KUKA KRL program: EPS_2_25362_MH4A_A_20251103083058.src

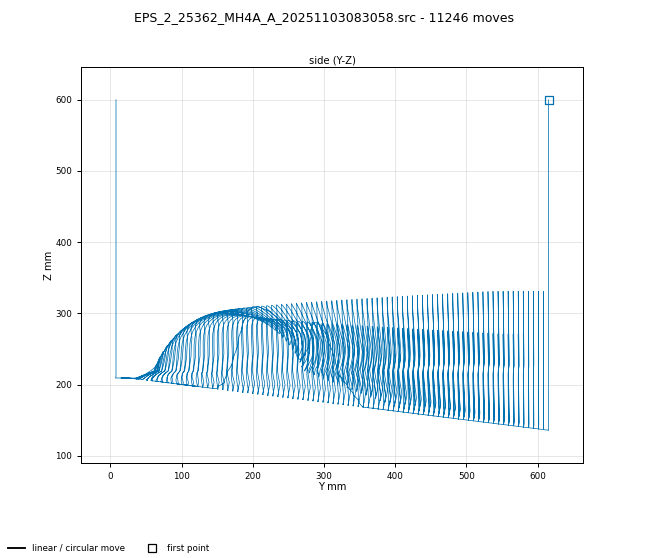
[picture p0: tool path of EPS_2_25362_MH4A_A_20251103083058.src, 11246 of 11248 moves have a stored position in this frame; points joined in program order, loops and branches not executed]
&ACCESS RVP
&REL 4
&COMMENT QRS 19112012
&PARAM EDITMASK = *
DEF PART()
EXT BAS (BAS_COMMAND :IN,REAL :IN )
INT I
BAS (#INITMOV,0 )

;KUKA QRS Post kuka4.cps  Date:22-06-2017 !

File_ID=2901

QRS_PRE_INIT()

;Init var - Until changes are made in qrs_pre_init
Outlet_Square_prg=0
Inlet_1_Square_prg=0
Inlet_2_Square_prg=0
Inlet_3_Square_prg=0
Inlet_4_Square_prg=0
Inlet_5_Square_prg=0

Outlet_1={X 0.000, Y 537.380, Z 230.500, B 0.000, E1 0.000 }
Inlet_1={X 0.000, Y 549.320, Z 220.500, B 0.000, E1 270.000 }
Outlet_1_type=201
Inlet_1_type=101
;QRS#1=Sidecore dimensions
;QRS#2=200-8" PVC SDR 35
;QRS#3=100-4" PVC SDR 28
;QRS#4=
;QRS#5=
;QRS#6=
;QRS#7=
;QRS#8=
;QRS#9=12-08 PSX
;QRS#10=8QRS PSX
;QRS#11=
;QRS#12=
;QRS#13=
;QRS#14=
;QRS#15=
;QRS#16=1220x127x610 2'
;QRS#17=EPS Height
;QRS#18=331
;QRS#19=*
;QRS#20= UPDATED VERSION 22-06-2017
;QRS#21=*
Outlet_Square=0100
Inlet_1_Square=045
Inlet_2_Square=0
Inlet_3_Square=0
Inlet_4_Square=0
Inlet_5_Square=0
Mill_Square=1
Outlet_Square_Prg=204
Inlet_1_Square_prg=201

QRS_INIT()

$ADVANCE=5

; T1
PTP {E1 173.59,E2 173.59}
PTP {X 0,Y 615.51,A -85,B 0,C 180,E1 173.59,E2 173.59,E3 0,E4 0,E5 0,E6 0}
QRS_SPEED_INIT()
LIN {X 0,Y 615.51,Z 600,A -85,B 0,C 180,E1 173.59,E2 173.59,E3 0,E4 0,E5 0,E6 0} C_VEL
LIN {X 0,Y 615.51,Z 145.871,A -85,B 0,C 180,E1 173.59,E2 173.59} C_VEL
LIN {X 0,Y 615.51,Z 137.691,A -85,B 0,C 180,E1 173.59,E2 173.59} C_VEL
LIN {X 0,Y 615.491,Z 135.691,A -85,B 0,C 180,E1 173.404,E2 173.404} C_VEL
LIN {X 0,Y 615.484,Z 135.694,A -85,B 0,C 180,E1 170.801,E2 170.801} C_VEL
LIN {X 0,Y 615.456,Z 135.696,A -85,B 0,C 180,E1 168.139,E2 168.139} C_VEL
LIN {X 0,Y 615.487,Z 135.702,A -85,B 0,C 180,E1 165.451,E2 165.451} C_VEL
LIN {X 0,Y 615.449,Z 135.697,A -85,B 0,C 180,E1 162.728,E2 162.728} C_VEL
LIN {X 0,Y 615.489,Z 135.692,A -85,B 0,C 180,E1 159.967,E2 159.967} C_VEL
LIN {X 0,Y 615.484,Z 135.699,A -85,B 0,C 180,E1 157.155,E2 157.155} C_VEL
LIN {X 0,Y 615.453,Z 135.696,A -85,B 0,C 180,E1 154.434,E2 154.434} C_VEL
LIN {X 0,Y 615.456,Z 135.699,A -85,B 0,C 180,E1 151.552,E2 151.552} C_VEL
LIN {X 0,Y 615.471,Z 135.698,A -85,B 0,C 180,E1 148.913,E2 148.913} C_VEL
LIN {X 0,Y 615.488,Z 135.688,A -85,B 0,C 180,E1 145.978,E2 145.978} C_VEL
LIN {X 0,Y 615.484,Z 135.703,A -85,B 0,C 180,E1 143.575,E2 143.575} C_VEL
LIN {X 0,Y 615.444,Z 135.698,A -85,B 0,C 180,E1 140.94,E2 140.94} C_VEL
LIN {X 0,Y 615.498,Z 135.7,A -85,B 0,C 180,E1 138.527,E2 138.527} C_VEL
LIN {X 0,Y 615.464,Z 135.694,A -85,B 0,C 180,E1 135.848,E2 135.848} C_VEL
LIN {X 0,Y 615.479,Z 135.693,A -85,B 0,C 180,E1 133.046,E2 133.046} C_VEL
LIN {X 0,Y 615.491,Z 135.7,A -85,B 0,C 180,E1 130.089,E2 130.089} C_VEL
LIN {X 0,Y 615.45,Z 135.7,A -85,B 0,C 180,E1 127.243,E2 127.243} C_VEL
LIN {X 0,Y 615.484,Z 135.692,A -85,B 0,C 180,E1 124.7,E2 124.7} C_VEL
LIN {X 0,Y 615.47,Z 135.694,A -85,B 0,C 180,E1 122.328,E2 122.328} C_VEL
LIN {X 0,Y 615.479,Z 135.696,A -85,B 0,C 180,E1 119.793,E2 119.793} C_VEL
LIN {X 0,Y 615.498,Z 135.691,A -85,B 0,C 180,E1 117.047,E2 117.047} C_VEL
LIN {X 0,Y 615.435,Z 135.7,A -85,B 0,C 180,E1 114.273,E2 114.273} C_VEL
LIN {X 0,Y 615.495,Z 135.693,A -85,B 0,C 180,E1 111.43,E2 111.43} C_VEL
LIN {X 0,Y 615.482,Z 135.696,A -85,B 0,C 180,E1 108.603,E2 108.603} C_VEL
LIN {X 0,Y 615.47,Z 135.692,A -85,B 0,C 180,E1 105.904,E2 105.904} C_VEL
LIN {X 0,Y 615.484,Z 135.7,A -85,B 0,C 180,E1 103.2,E2 103.2} C_VEL
LIN {X 0,Y 615.442,Z 135.7,A -85,B 0,C 180,E1 100.527,E2 100.527} C_VEL
LIN {X 0,Y 615.493,Z 135.691,A -85,B 0,C 180,E1 97.874,E2 97.874} C_VEL
LIN {X 0,Y 615.483,Z 135.695,A -85,B 0,C 180,E1 95.24,E2 95.24} C_VEL
LIN {X 0,Y 615.461,Z 135.695,A -85,B 0,C 180,E1 92.617,E2 92.617} C_VEL
LIN {X 0,Y 615.486,Z 135.699,A -85,B 0,C 180,E1 89.999,E2 89.999} C_VEL
LIN {X 0,Y 615.446,Z 135.697,A -85,B 0,C 180,E1 87.381,E2 87.381} C_VEL
LIN {X 0,Y 615.491,Z 135.699,A -85,B 0,C 180,E1 84.758,E2 84.758} C_VEL
LIN {X 0,Y 615.488,Z 135.689,A -85,B 0,C 180,E1 82.123,E2 82.123} C_VEL
LIN {X 0,Y 615.466,Z 135.698,A -85,B 0,C 180,E1 79.472,E2 79.472} C_VEL
LIN {X 0,Y 615.458,Z 135.7,A -85,B 0,C 180,E1 76.797,E2 76.797} C_VEL
LIN {X 0,Y 615.461,Z 135.695,A -85,B 0,C 180,E1 74.093,E2 74.093} C_VEL
LIN {X 0,Y 615.492,Z 135.7,A -85,B 0,C 180,E1 71.353,E2 71.353} C_VEL
LIN {X 0,Y 615.492,Z 135.689,A -85,B 0,C 180,E1 68.567,E2 68.567} C_VEL
LIN {X 0,Y 615.446,Z 135.698,A -85,B 0,C 180,E1 65.725,E2 65.725} C_VEL
LIN {X 0,Y 615.485,Z 135.697,A -85,B 0,C 180,E1 62.822,E2 62.822} C_VEL
LIN {X 0,Y 615.462,Z 135.696,A -85,B 0,C 180,E1 60.21,E2 60.21} C_VEL
LIN {X 0,Y 615.479,Z 135.693,A -85,B 0,C 180,E1 57.541,E2 57.541} C_VEL
LIN {X 0,Y 615.496,Z 135.688,A -85,B 0,C 180,E1 55.185,E2 55.185} C_VEL
LIN {X 0,Y 615.471,Z 135.7,A -85,B 0,C 180,E1 52.756,E2 52.756} C_VEL
LIN {X 0,Y 615.459,Z 135.7,A -85,B 0,C 180,E1 49.914,E2 49.914} C_VEL
LIN {X 0,Y 615.494,Z 135.693,A -85,B 0,C 180,E1 47.647,E2 47.647} C_VEL
LIN {X 0,Y 615.478,Z 135.695,A -85,B 0,C 180,E1 44.93,E2 44.93} C_VEL
LIN {X 0,Y 615.463,Z 135.695,A -85,B 0,C 180,E1 42.355,E2 42.355} C_VEL
LIN {X 0,Y 615.491,Z 135.695,A -85,B 0,C 180,E1 39.75,E2 39.75} C_VEL
LIN {X 0,Y 615.441,Z 135.699,A -85,B 0,C 180,E1 36.93,E2 36.93} C_VEL
LIN {X 0,Y 615.479,Z 135.698,A -85,B 0,C 180,E1 34.699,E2 34.699} C_VEL
LIN {X 0,Y 615.481,Z 135.692,A -85,B 0,C 180,E1 32.329,E2 32.329} C_VEL
LIN {X 0,Y 615.493,Z 135.842,A -85,B 0,C 180,E1 29.746,E2 29.746} C_VEL
LIN {X 0,Y 615.494,Z 144.518,A -85,B 0,C 180,E1 27.045,E2 27.045} C_VEL
LIN {X 0,Y 615.484,Z 153.55,A -85,B 0,C 180,E1 24.272,E2 24.272} C_VEL
LIN {X 0,Y 615.429,Z 162.982,A -85,B 0,C 180,E1 21.434,E2 21.434} C_VEL
LIN {X 0,Y 615.491,Z 172.39,A -85,B 0,C 180,E1 18.646,E2 18.646} C_VEL
LIN {X 0,Y 615.466,Z 181.817,A -85,B 0,C 180,E1 15.906,E2 15.906} C_VEL
LIN {X 0,Y 615.484,Z 191.214,A -85,B 0,C 180,E1 13.201,E2 13.201} C_VEL
LIN {X 0,Y 615.49,Z 200.624,A -85,B 0,C 180,E1 10.527,E2 10.527} C_VEL
LIN {X 0,Y 615.463,Z 210.021,A -85,B 0,C 180,E1 7.876,E2 7.876} C_VEL
LIN {X 0,Y 615.497,Z 214.015,A -85,B 0,C 180,E1 6.761,E2 6.761} C_VEL
LIN {X 0,Y 615.497,Z 223.447,A -85,B 0,C 180,E1 6.474,E2 6.474} C_VEL
LIN {X 0,Y 615.451,Z 232.476,A -85,B 0,C 180,E1 6.063,E2 6.063} C_VEL
LIN {X 0,Y 615.437,Z 240.486,A -85,B 0,C 180,E1 5.57,E2 5.57} C_VEL
LIN {X 0,Y 615.483,Z 248.518,A -85,B 0,C 180,E1 4.913,E2 4.913} C_VEL
LIN {X 0,Y 615.497,Z 254.668,A -85,B 0,C 180,E1 4.256,E2 4.256} C_VEL
LIN {X 0,Y 615.497,Z 259.516,A -85,B 0,C 180,E1 3.601,E2 3.601} C_VEL
LIN {X 0,Y 615.498,Z 263.25,A -85,B 0,C 180,E1 2.945,E2 2.945} C_VEL
LIN {X 0,Y 615.498,Z 267.23,A -85,B 0,C 180,E1 1.963,E2 1.963} C_VEL
LIN {X 0,Y 615.496,Z 268.964,A -85,B 0,C 180,E1 1.309,E2 1.309} C_VEL
LIN {X 0,Y 615.496,Z 270.004,A -85,B 0,C 180,E1 0.654,E2 0.654} C_VEL
LIN {X 0,Y 615.494,Z 270.384,A -85,B 0,C 180,E1 0,E2 0} C_VEL
LIN {X 0,Y 615.496,Z 270.105,A -85,B 0,C 180,E1 -0.654,E2 -0.654} C_VEL
LIN {X 0,Y 615.497,Z 269.165,A -85,B 0,C 180,E1 -1.309,E2 -1.309} C_VEL
LIN {X 0,Y 615.496,Z 267.536,A -85,B 0,C 180,E1 -1.963,E2 -1.963} C_VEL
LIN {X 0,Y 615.498,Z 263.663,A -85,B 0,C 180,E1 -2.945,E2 -2.945} C_VEL
LIN {X 0,Y 615.5,Z 259.011,A -85,B 0,C 180,E1 -3.765,E2 -3.765} C_VEL
LIN {X 0,Y 615.498,Z 254.03,A -85,B 0,C 180,E1 -4.42,E2 -4.42} C_VEL
LIN {X 0,Y 615.467,Z 247.759,A -85,B 0,C 180,E1 -5.077,E2 -5.077} C_VEL
LIN {X 0,Y 615.43,Z 240.602,A -85,B 0,C 180,E1 -5.653,E2 -5.653} C_VEL
LIN {X 0,Y 615.448,Z 232.615,A -85,B 0,C 180,E1 -6.146,E2 -6.146} C_VEL
LIN {X 0,Y 615.488,Z 223.109,A -85,B 0,C 180,E1 -6.576,E2 -6.576} C_VEL
LIN {X 0,Y 615.489,Z 213.97,A -85,B 0,C 180,E1 -6.856,E2 -6.856} C_VEL
LIN {X 0,Y 615.458,Z 204.468,A -85,B 0,C 180,E1 -9.531,E2 -9.531} C_VEL
LIN {X 0,Y 615.485,Z 195.061,A -85,B 0,C 180,E1 -12.195,E2 -12.195} C_VEL
LIN {X 0,Y 615.482,Z 185.648,A -85,B 0,C 180,E1 -14.887,E2 -14.887} C_VEL
LIN {X 0,Y 615.461,Z 176.24,A -85,B 0,C 180,E1 -17.614,E2 -17.614} C_VEL
LIN {X 0,Y 615.468,Z 167.99,A -85,B 0,C 180,E1 -20.034,E2 -20.034} C_VEL
LIN {X 0,Y 615.44,Z 158.569,A -85,B 0,C 180,E1 -22.847,E2 -22.847} C_VEL
LIN {X 0,Y 615.439,Z 151.492,A -85,B 0,C 180,E1 -24.994,E2 -24.994} C_VEL
LIN {X 0,Y 615.496,Z 143.116,A -85,B 0,C 180,E1 -27.545,E2 -27.545} C_VEL
LIN {X 0,Y 615.489,Z 135.697,A -85,B 0,C 180,E1 -29.794,E2 -29.794} C_VEL
LIN {X 0,Y 615.488,Z 135.698,A -85,B 0,C 180,E1 -32.458,E2 -32.458} C_VEL
LIN {X 0,Y 615.493,Z 135.7,A -85,B 0,C 180,E1 -34.815,E2 -34.815} C_VEL
LIN {X 0,Y 615.491,Z 135.699,A -85,B 0,C 180,E1 -37.242,E2 -37.242} C_VEL
LIN {X 0,Y 615.489,Z 135.698,A -85,B 0,C 180,E1 -40.088,E2 -40.088} C_VEL
LIN {X 0,Y 615.487,Z 135.7,A -85,B 0,C 180,E1 -42.353,E2 -42.353} C_VEL
LIN {X 0,Y 615.485,Z 135.698,A -85,B 0,C 180,E1 -45.069,E2 -45.069} C_VEL
LIN {X 0,Y 615.494,Z 135.701,A -85,B 0,C 180,E1 -47.919,E2 -47.919} C_VEL
LIN {X 0,Y 615.487,Z 135.701,A -85,B 0,C 180,E1 -50.249,E2 -50.249} C_VEL
LIN {X 0,Y 615.483,Z 135.698,A -85,B 0,C 180,E1 -53.064,E2 -53.064} C_VEL
LIN {X 0,Y 615.496,Z 135.696,A -85,B 0,C 180,E1 -55.299,E2 -55.299} C_VEL
LIN {X 0,Y 615.494,Z 135.699,A -85,B 0,C 180,E1 -57.669,E2 -57.669} C_VEL
LIN {X 0,Y 615.479,Z 135.7,A -85,B 0,C 180,E1 -60.207,E2 -60.207} C_VEL
LIN {X 0,Y 615.498,Z 135.696,A -85,B 0,C 180,E1 -62.953,E2 -62.953} C_VEL
LIN {X 0,Y 615.472,Z 135.812,A -85,B 0,C 180,E1 -63.76,E2 -63.76} C_VEL
LIN {X 0,Y 615.493,Z 150.876,A -85,B 0,C 180,E1 -66.443,E2 -66.443} C_VEL
LIN {X 0,Y 615.49,Z 167.065,A -85,B 0,C 180,E1 -69.269,E2 -69.269} C_VEL
LIN {X 0,Y 615.477,Z 183.238,A -85,B 0,C 180,E1 -72.042,E2 -72.042} C_VEL
LIN {X 0,Y 615.485,Z 199.394,A -85,B 0,C 180,E1 -74.773,E2 -74.773} C_VEL
LIN {X 0,Y 615.491,Z 215.538,A -85,B 0,C 180,E1 -77.469,E2 -77.469} C_VEL
LIN {X 0,Y 615.493,Z 220.864,A -85,B 0,C 180,E1 -78.326,E2 -78.326} C_VEL
LIN {X 0,Y 615.486,Z 234.201,A -85,B 0,C 180,E1 -78.556,E2 -78.556} C_VEL
LIN {X 0,Y 615.476,Z 247.357,A -85,B 0,C 180,E1 -78.923,E2 -78.923} C_VEL
LIN {X 0,Y 615.486,Z 259.131,A -85,B 0,C 180,E1 -79.383,E2 -79.383} C_VEL
LIN {X 0,Y 615.483,Z 270.56,A -85,B 0,C 180,E1 -79.971,E2 -79.971} C_VEL
LIN {X 0,Y 615.499,Z 282.008,A -85,B 0,C 180,E1 -80.718,E2 -80.718} C_VEL
LIN {X 0,Y 615.498,Z 291.247,A -85,B 0,C 180,E1 -81.463,E2 -81.463} C_VEL
LIN {X 0,Y 615.5,Z 299.645,A -85,B 0,C 180,E1 -82.289,E2 -82.289} C_VEL
LIN {X 0,Y 615.497,Z 307.688,A -85,B 0,C 180,E1 -83.258,E2 -83.258} C_VEL
LIN {X 0,Y 615.499,Z 313.417,A -85,B 0,C 180,E1 -84.101,E2 -84.101} C_VEL
LIN {X 0,Y 615.496,Z 318.868,A -85,B 0,C 180,E1 -85.086,E2 -85.086} C_VEL
LIN {X 0,Y 615.497,Z 323.137,A -85,B 0,C 180,E1 -86.071,E2 -86.071} C_VEL
LIN {X 0,Y 615.494,Z 325.396,A -85,B 0,C 180,E1 -86.726,E2 -86.726} C_VEL
LIN {X 0,Y 615.497,Z 327.23,A -85,B 0,C 180,E1 -87.381,E2 -87.381} C_VEL
LIN {X 0,Y 615.5,Z 328.606,A -85,B 0,C 180,E1 -88.036,E2 -88.036} C_VEL
LIN {X 0,Y 615.496,Z 330.173,A -85,B 0,C 180,E1 -89.345,E2 -89.345} C_VEL
LIN {X 0,Y 615.494,Z 330.389,A -85,B 0,C 180,E1 -89.999,E2 -89.999} C_VEL
LIN {X 0,Y 615.495,Z 329.581,A -85,B 0,C 180,E1 -91.308,E2 -91.308} C_VEL
LIN {X 0,Y 615.5,Z 328.609,A -85,B 0,C 180,E1 -91.962,E2 -91.962} C_VEL
LIN {X 0,Y 615.497,Z 327.236,A -85,B 0,C 180,E1 -92.617,E2 -92.617} C_VEL
LIN {X 0,Y 615.496,Z 324.353,A -85,B 0,C 180,E1 -93.6,E2 -93.6} C_VEL
LIN {X 0,Y 615.498,Z 320.446,A -85,B 0,C 180,E1 -94.583,E2 -94.583} C_VEL
LIN {X 0,Y 615.499,Z 315.411,A -85,B 0,C 180,E1 -95.569,E2 -95.569} C_VEL
LIN {X 0,Y 615.496,Z 308.87,A -85,B 0,C 180,E1 -96.583,E2 -96.583} C_VEL
LIN {X 0,Y 615.497,Z 301.143,A -85,B 0,C 180,E1 -97.544,E2 -97.544} C_VEL
LIN {X 0,Y 615.498,Z 293.057,A -85,B 0,C 180,E1 -98.37,E2 -98.37} C_VEL
LIN {X 0,Y 615.499,Z 283.183,A -85,B 0,C 180,E1 -99.197,E2 -99.197} C_VEL
LIN {X 0,Y 615.485,Z 272.002,A -85,B 0,C 180,E1 -99.944,E2 -99.944} C_VEL
LIN {X 0,Y 615.489,Z 261.047,A -85,B 0,C 180,E1 -100.526,E2 -100.526} C_VEL
LIN {X 0,Y 615.476,Z 248.567,A -85,B 0,C 180,E1 -101.038,E2 -101.038} C_VEL
LIN {X 0,Y 615.485,Z 236.118,A -85,B 0,C 180,E1 -101.4,E2 -101.4} C_VEL
LIN {X 0,Y 615.492,Z 222.551,A -85,B 0,C 180,E1 -101.651,E2 -101.651} C_VEL
LIN {X 0,Y 615.494,Z 220.593,A -85,B 0,C 180,E1 -101.692,E2 -101.692} C_VEL
LIN {X 0,Y 615.487,Z 203.445,A -85,B 0,C 180,E1 -104.548,E2 -104.548} C_VEL
LIN {X 0,Y 615.493,Z 186.28,A -85,B 0,C 180,E1 -107.44,E2 -107.44} C_VEL
LIN {X 0,Y 615.478,Z 169.601,A -85,B 0,C 180,E1 -110.294,E2 -110.294} C_VEL
LIN {X 0,Y 615.493,Z 153.925,A -85,B 0,C 180,E1 -113.02,E2 -113.02} C_VEL
LIN {X 0,Y 615.498,Z 138.737,A -85,B 0,C 180,E1 -115.714,E2 -115.714} C_VEL
LIN {X 0,Y 615.456,Z 135.697,A -85,B 0,C 180,E1 -116.284,E2 -116.284} C_VEL
LIN {X 0,Y 615.456,Z 135.699,A -85,B 0,C 180,E1 -118.658,E2 -118.658} C_VEL
LIN {X 0,Y 615.48,Z 135.695,A -85,B 0,C 180,E1 -121.084,E2 -121.084} C_VEL
LIN {X 0,Y 615.467,Z 135.694,A -85,B 0,C 180,E1 -123.531,E2 -123.531} C_VEL
LIN {X 0,Y 615.488,Z 135.701,A -85,B 0,C 180,E1 -125.833,E2 -125.833} C_VEL
LIN {X 0,Y 615.463,Z 135.695,A -85,B 0,C 180,E1 -128.068,E2 -128.068} C_VEL
LIN {X 0,Y 615.481,Z 135.698,A -85,B 0,C 180,E1 -130.605,E2 -130.605} C_VEL
LIN {X 0,Y 615.442,Z 135.698,A -85,B 0,C 180,E1 -133.247,E2 -133.247} C_VEL
LIN {X 0,Y 615.49,Z 135.697,A -85,B 0,C 180,E1 -136,E2 -136} C_VEL
LIN {X 0,Y 615.486,Z 135.695,A -85,B 0,C 180,E1 -138.903,E2 -138.903} C_VEL
LIN {X 0,Y 615.477,Z 135.699,A -85,B 0,C 180,E1 -141.095,E2 -141.095} C_VEL
LIN {X 0,Y 615.441,Z 135.699,A -85,B 0,C 180,E1 -143.572,E2 -143.572} C_VEL
LIN {X 0,Y 615.465,Z 135.695,A -85,B 0,C 180,E1 -146.466,E2 -146.466} C_VEL
LIN {X 0,Y 615.482,Z 135.698,A -85,B 0,C 180,E1 -149.08,E2 -149.08} C_VEL
LIN {X 0,Y 615.478,Z 135.691,A -85,B 0,C 180,E1 -151.548,E2 -151.548} C_VEL
LIN {X 0,Y 615.48,Z 135.701,A -85,B 0,C 180,E1 -154.429,E2 -154.429} C_VEL
LIN {X 0,Y 615.448,Z 135.7,A -85,B 0,C 180,E1 -156.442,E2 -156.442} C_VEL
LIN {X 0,Y 615.441,Z 135.699,A -85,B 0,C 180,E1 -158.566,E2 -158.566} C_VEL
LIN {X 0,Y 615.492,Z 135.692,A -85,B 0,C 180,E1 -161.389,E2 -161.389} C_VEL
LIN {X 0,Y 615.486,Z 135.695,A -85,B 0,C 180,E1 -164.095,E2 -164.095} C_VEL
LIN {X 0,Y 615.456,Z 135.695,A -85,B 0,C 180,E1 -166.798,E2 -166.798} C_VEL
LIN {X 0,Y 615.481,Z 135.702,A -85,B 0,C 180,E1 -169.473,E2 -169.473} C_VEL
LIN {X 0,Y 615.45,Z 135.697,A -85,B 0,C 180,E1 -172.124,E2 -172.124} C_VEL
LIN {X 0,Y 615.486,Z 135.694,A -85,B 0,C 180,E1 -174.759,E2 -174.759} C_VEL
LIN {X 0,Y 615.489,Z 135.691,A -85,B 0,C 180,E1 -177.382,E2 -177.382} C_VEL
LIN {X 0,Y 615.454,Z 135.698,A -85,B 0,C 180,E1 -180,E2 -180} C_VEL
LIN {X 0,Y 615.466,Z 135.701,A -85,B 0,C 180,E1 -182.618,E2 -182.618} C_VEL
LIN {X 0,Y 615.464,Z 135.694,A -85,B 0,C 180,E1 -185.241,E2 -185.241} C_VEL
LIN {X 0,Y 615.491,Z 135.691,A -85,B 0,C 180,E1 -186.596,E2 -186.596} C_VEL
LIN {X 0,Y 614.805,Z 135.838,A -85,B 0,C 180,E1 -187.142,E2 -187.142} C_VEL
LIN {X 0,Y 611.966,Z 136.258,A -85,B 0,C 180,E1 -188.028,E2 -188.028} C_VEL
LIN {X 0,Y 609.577,Z 136.568,A -85,B 0,C 180,E1 -188.74,E2 -188.74} C_VEL
LIN {X 0,Y 608.543,Z 136.684,A -85,B 0,C 180,E1 -189.29,E2 -189.29} C_VEL
LIN {X 0,Y 608.453,Z 136.693,A -85,B 0,C 180,E1 -189.476,E2 -189.476} C_VEL
LIN {X 0,Y 608.44,Z 136.692,A -85,B 0,C 180,E1 -192,E2 -192} C_VEL
LIN {X 0,Y 608.462,Z 136.695,A -85,B 0,C 180,E1 -194.721,E2 -194.721} C_VEL
LIN {X 0,Y 608.431,Z 136.695,A -85,B 0,C 180,E1 -197.477,E2 -197.477} C_VEL
LIN {X 0,Y 608.462,Z 136.69,A -85,B 0,C 180,E1 -200.274,E2 -200.274} C_VEL
LIN {X 0,Y 608.48,Z 136.688,A -85,B 0,C 180,E1 -202.486,E2 -202.486} C_VEL
LIN {X 0,Y 608.446,Z 136.698,A -85,B 0,C 180,E1 -204.571,E2 -204.571} C_VEL
LIN {X 0,Y 608.422,Z 136.695,A -85,B 0,C 180,E1 -207.519,E2 -207.519} C_VEL
LIN {X 0,Y 608.471,Z 136.692,A -85,B 0,C 180,E1 -209.975,E2 -209.975} C_VEL
LIN {X 0,Y 608.449,Z 136.696,A -85,B 0,C 180,E1 -212.88,E2 -212.88} C_VEL
LIN {X 0,Y 608.443,Z 136.693,A -85,B 0,C 180,E1 -215.278,E2 -215.278} C_VEL
LIN {X 0,Y 608.463,Z 136.694,A -85,B 0,C 180,E1 -218.242,E2 -218.242} C_VEL
LIN {X 0,Y 608.455,Z 136.696,A -85,B 0,C 180,E1 -221.344,E2 -221.344} C_VEL
LIN {X 0,Y 608.456,Z 136.69,A -85,B 0,C 180,E1 -223.871,E2 -223.871} C_VEL
LIN {X 0,Y 608.47,Z 136.693,A -85,B 0,C 180,E1 -226.691,E2 -226.691} C_VEL
LIN {X 0,Y 608.474,Z 136.693,A -85,B 0,C 180,E1 -229.669,E2 -229.669} C_VEL
LIN {X 0,Y 608.452,Z 136.693,A -85,B 0,C 180,E1 -232.844,E2 -232.844} C_VEL
LIN {X 0,Y 608.46,Z 136.69,A -85,B 0,C 180,E1 -235.532,E2 -235.532} C_VEL
LIN {X 0,Y 608.458,Z 136.693,A -85,B 0,C 180,E1 -237.907,E2 -237.907} C_VEL
LIN {X 0,Y 608.464,Z 136.692,A -85,B 0,C 180,E1 -240.222,E2 -240.222} C_VEL
LIN {X 0,Y 608.48,Z 136.688,A -85,B 0,C 180,E1 -242.793,E2 -242.793} C_VEL
LIN {X 0,Y 608.43,Z 136.695,A -85,B 0,C 180,E1 -245.429,E2 -245.429} C_VEL
LIN {X 0,Y 608.463,Z 136.697,A -85,B 0,C 180,E1 -248.31,E2 -248.31} C_VEL
LIN {X 0,Y 608.467,Z 136.691,A -85,B 0,C 180,E1 -251.285,E2 -251.285} C_VEL
LIN {X 0,Y 608.449,Z 136.692,A -85,B 0,C 180,E1 -253.907,E2 -253.907} C_VEL
LIN {X 0,Y 608.458,Z 136.697,A -85,B 0,C 180,E1 -256.645,E2 -256.645} C_VEL
LIN {X 0,Y 608.421,Z 136.695,A -85,B 0,C 180,E1 -259.351,E2 -259.351} C_VEL
LIN {X 0,Y 608.481,Z 136.69,A -85,B 0,C 180,E1 -262.034,E2 -262.034} C_VEL
LIN {X 0,Y 608.464,Z 136.691,A -85,B 0,C 180,E1 -264.699,E2 -264.699} C_VEL
LIN {X 0,Y 608.455,Z 136.691,A -85,B 0,C 180,E1 -267.353,E2 -267.353} C_VEL
LIN {X 0,Y 608.477,Z 136.693,A -85,B 0,C 180,E1 -270.001,E2 -270.001} C_VEL
LIN {X 0,Y 608.442,Z 136.692,A -85,B 0,C 180,E1 -272.649,E2 -272.649} C_VEL
LIN {X 0,Y 608.471,Z 136.694,A -85,B 0,C 180,E1 -275.303,E2 -275.303} C_VEL
LIN {X 0,Y 608.48,Z 136.688,A -85,B 0,C 180,E1 -277.968,E2 -277.968} C_VEL
LIN {X 0,Y 608.449,Z 136.691,A -85,B 0,C 180,E1 -280.945,E2 -280.945} C_VEL
LIN {X 0,Y 608.437,Z 136.697,A -85,B 0,C 180,E1 -283.358,E2 -283.358} C_VEL
LIN {X 0,Y 608.437,Z 136.692,A -85,B 0,C 180,E1 -286.095,E2 -286.095} C_VEL
LIN {X 0,Y 608.461,Z 136.693,A -85,B 0,C 180,E1 -288.87,E2 -288.87} C_VEL
LIN {X 0,Y 608.47,Z 136.692,A -85,B 0,C 180,E1 -291.692,E2 -291.692} C_VEL
LIN {X 0,Y 608.432,Z 136.693,A -85,B 0,C 180,E1 -294.573,E2 -294.573} C_VEL
LIN {X 0,Y 608.461,Z 136.694,A -85,B 0,C 180,E1 -297.204,E2 -297.204} C_VEL
LIN {X 0,Y 608.452,Z 136.693,A -85,B 0,C 180,E1 -299.969,E2 -299.969} C_VEL
LIN {X 0,Y 608.455,Z 136.69,A -85,B 0,C 180,E1 -302.88,E2 -302.88} C_VEL
LIN {X 0,Y 608.44,Z 136.698,A -85,B 0,C 180,E1 -305.279,E2 -305.279} C_VEL
LIN {X 0,Y 608.414,Z 136.695,A -85,B 0,C 180,E1 -307.751,E2 -307.751} C_VEL
LIN {X 0,Y 608.439,Z 136.699,A -85,B 0,C 180,E1 -310.327,E2 -310.327} C_VEL
LIN {X 0,Y 608.439,Z 136.692,A -85,B 0,C 180,E1 -312.962,E2 -312.962} C_VEL
LIN {X 0,Y 608.448,Z 136.694,A -85,B 0,C 180,E1 -315.738,E2 -315.738} C_VEL
LIN {X 0,Y 608.464,Z 136.695,A -85,B 0,C 180,E1 -318.658,E2 -318.658} C_VEL
LIN {X 0,Y 608.405,Z 136.696,A -85,B 0,C 180,E1 -321.407,E2 -321.407} C_VEL
LIN {X 0,Y 608.45,Z 136.697,A -85,B 0,C 180,E1 -323.955,E2 -323.955} C_VEL
LIN {X 0,Y 608.448,Z 136.691,A -85,B 0,C 180,E1 -326.328,E2 -326.328} C_VEL
LIN {X 0,Y 608.451,Z 136.696,A -85,B 0,C 180,E1 -328.733,E2 -328.733} C_VEL
LIN {X 0,Y 608.482,Z 136.743,A -85,B 0,C 180,E1 -330.159,E2 -330.159} C_VEL
LIN {X 0,Y 608.485,Z 145.123,A -85,B 0,C 180,E1 -332.792,E2 -332.792} C_VEL
LIN {X 0,Y 608.44,Z 153.666,A -85,B 0,C 180,E1 -335.428,E2 -335.428} C_VEL
LIN {X 0,Y 608.412,Z 163.13,A -85,B 0,C 180,E1 -338.306,E2 -338.306} C_VEL
LIN {X 0,Y 608.429,Z 171.411,A -85,B 0,C 180,E1 -340.779,E2 -340.779} C_VEL
LIN {X 0,Y 608.444,Z 180.597,A -85,B 0,C 180,E1 -343.48,E2 -343.48} C_VEL
LIN {X 0,Y 608.444,Z 190.398,A -85,B 0,C 180,E1 -346.32,E2 -346.32} C_VEL
LIN {X 0,Y 608.422,Z 200.004,A -85,B 0,C 180,E1 -349.069,E2 -349.069} C_VEL
LIN {X 0,Y 608.45,Z 209.27,A -85,B 0,C 180,E1 -351.698,E2 -351.698} C_VEL
LIN {X 0,Y 608.427,Z 214.373,A -85,B 0,C 180,E1 -353.138,E2 -353.138} C_VEL
LIN {X 0,Y 608.475,Z 225.425,A -85,B 0,C 180,E1 -353.505,E2 -353.505} C_VEL
LIN {X 0,Y 608.403,Z 234.473,A -85,B 0,C 180,E1 -353.949,E2 -353.949} C_VEL
LIN {X 0,Y 608.407,Z 243.253,A -85,B 0,C 180,E1 -354.531,E2 -354.531} C_VEL
LIN {X 0,Y 608.455,Z 249.028,A -85,B 0,C 180,E1 -355.03,E2 -355.03} C_VEL
LIN {X 0,Y 608.443,Z 255.206,A -85,B 0,C 180,E1 -355.694,E2 -355.694} C_VEL
LIN {X 0,Y 608.451,Z 260.068,A -85,B 0,C 180,E1 -356.358,E2 -356.358} C_VEL
LIN {X 0,Y 608.452,Z 263.818,A -85,B 0,C 180,E1 -357.021,E2 -357.021} C_VEL
LIN {X 0,Y 608.443,Z 267.825,A -85,B 0,C 180,E1 -358.014,E2 -358.014} C_VEL
LIN {X 0,Y 608.448,Z 269.569,A -85,B 0,C 180,E1 -358.676,E2 -358.676} C_VEL
LIN {X 0,Y 608.439,Z 270.615,A -85,B 0,C 180,E1 -359.338,E2 -359.338} C_VEL
LIN {X 0,Y 608.434,Z 270.995,A -85,B 0,C 180,E1 -360,E2 -360} C_VEL
LIN {X 0,Y 608.438,Z 270.714,A -85,B 0,C 180,E1 -360.662,E2 -360.662} C_VEL
LIN {X 0,Y 608.449,Z 269.768,A -85,B 0,C 180,E1 -361.324,E2 -361.324} C_VEL
LIN {X 0,Y 608.442,Z 268.128,A -85,B 0,C 180,E1 -361.986,E2 -361.986} C_VEL
LIN {X 0,Y 608.429,Z 265.745,A -85,B 0,C 180,E1 -362.648,E2 -362.648} C_VEL
LIN {X 0,Y 608.452,Z 260.617,A -85,B 0,C 180,E1 -363.642,E2 -363.642} C_VEL
LIN {X 0,Y 608.451,Z 254.555,A -85,B 0,C 180,E1 -364.472,E2 -364.472} C_VEL
LIN {X 0,Y 608.429,Z 248.249,A -85,B 0,C 180,E1 -365.136,E2 -365.136} C_VEL
LIN {X 0,Y 608.41,Z 241.092,A -85,B 0,C 180,E1 -365.718,E2 -365.718} C_VEL
LIN {X 0,Y 608.406,Z 233.106,A -85,B 0,C 180,E1 -366.217,E2 -366.217} C_VEL
LIN {X 0,Y 608.483,Z 224.258,A -85,B 0,C 180,E1 -366.633,E2 -366.633} C_VEL
LIN {X 0,Y 608.422,Z 214.4,A -85,B 0,C 180,E1 -366.945,E2 -366.945} C_VEL
LIN {X 0,Y 608.397,Z 206.038,A -85,B 0,C 180,E1 -369.307,E2 -369.307} C_VEL
LIN {X 0,Y 608.422,Z 197.753,A -85,B 0,C 180,E1 -371.663,E2 -371.663} C_VEL
LIN {X 0,Y 608.448,Z 188.285,A -85,B 0,C 180,E1 -374.379,E2 -374.379} C_VEL
LIN {X 0,Y 608.445,Z 178.816,A -85,B 0,C 180,E1 -377.13,E2 -377.13} C_VEL
LIN {X 0,Y 608.427,Z 170.531,A -85,B 0,C 180,E1 -379.572,E2 -379.572} C_VEL
LIN {X 0,Y 608.434,Z 162.245,A -85,B 0,C 180,E1 -382.05,E2 -382.05} C_VEL
LIN {X 0,Y 608.438,Z 153.959,A -85,B 0,C 180,E1 -384.572,E2 -384.572} C_VEL
LIN {X 0,Y 608.486,Z 145.357,A -85,B 0,C 180,E1 -387.208,E2 -387.208} C_VEL
LIN {X 0,Y 608.484,Z 136.692,A -85,B 0,C 180,E1 -389.841,E2 -389.841} C_VEL
LIN {X 0,Y 608.453,Z 136.697,A -85,B 0,C 180,E1 -392.88,E2 -392.88} C_VEL
LIN {X 0,Y 608.445,Z 136.696,A -85,B 0,C 180,E1 -395.278,E2 -395.278} C_VEL
LIN {X 0,Y 608.478,Z 136.692,A -85,B 0,C 180,E1 -397.746,E2 -397.746} C_VEL
LIN {X 0,Y 608.449,Z 136.699,A -85,B 0,C 180,E1 -400.328,E2 -400.328} C_VEL
LIN {X 0,Y 608.469,Z 136.694,A -85,B 0,C 180,E1 -403.308,E2 -403.308} C_VEL
LIN {X 0,Y 608.469,Z 136.693,A -85,B 0,C 180,E1 -406.13,E2 -406.13} C_VEL
LIN {X 0,Y 608.45,Z 136.697,A -85,B 0,C 180,E1 -408.822,E2 -408.822} C_VEL
LIN {X 0,Y 608.46,Z 136.694,A -85,B 0,C 180,E1 -411.761,E2 -411.761} C_VEL
LIN {X 0,Y 608.448,Z 136.696,A -85,B 0,C 180,E1 -413.955,E2 -413.955} C_VEL
LIN {X 0,Y 608.448,Z 136.696,A -85,B 0,C 180,E1 -416.328,E2 -416.328} C_VEL
LIN {X 0,Y 608.452,Z 136.697,A -85,B 0,C 180,E1 -418.732,E2 -418.732} C_VEL
LIN {X 0,Y 608.465,Z 136.694,A -85,B 0,C 180,E1 -421.382,E2 -421.382} C_VEL
LIN {X 0,Y 608.447,Z 136.699,A -85,B 0,C 180,E1 -423.595,E2 -423.595} C_VEL
LIN {X 0,Y 608.551,Z 148.233,A -85,B 0,C 180,E1 -425.684,E2 -425.684} C_VEL
LIN {X 0,Y 608.529,Z 164.059,A -85,B 0,C 180,E1 -428.488,E2 -428.488} C_VEL
LIN {X 0,Y 608.517,Z 180.072,A -85,B 0,C 180,E1 -431.272,E2 -431.272} C_VEL
LIN {X 0,Y 608.486,Z 196.485,A -85,B 0,C 180,E1 -434.078,E2 -434.078} C_VEL
LIN {X 0,Y 608.459,Z 212.699,A -85,B 0,C 180,E1 -436.813,E2 -436.813} C_VEL
LIN {X 0,Y 608.475,Z 221.013,A -85,B 0,C 180,E1 -438.19,E2 -438.19} C_VEL
LIN {X 0,Y 608.534,Z 234.314,A -85,B 0,C 180,E1 -438.423,E2 -438.423} C_VEL
LIN {X 0,Y 608.52,Z 247.201,A -85,B 0,C 180,E1 -438.785,E2 -438.785} C_VEL
LIN {X 0,Y 608.509,Z 259.275,A -85,B 0,C 180,E1 -439.26,E2 -439.26} C_VEL
LIN {X 0,Y 608.493,Z 270.74,A -85,B 0,C 180,E1 -439.854,E2 -439.854} C_VEL
LIN {X 0,Y 608.504,Z 282.239,A -85,B 0,C 180,E1 -440.61,E2 -440.61} C_VEL
LIN {X 0,Y 608.472,Z 291.525,A -85,B 0,C 180,E1 -441.363,E2 -441.363} C_VEL
LIN {X 0,Y 608.456,Z 299.981,A -85,B 0,C 180,E1 -442.199,E2 -442.199} C_VEL
LIN {X 0,Y 608.463,Z 308.228,A -85,B 0,C 180,E1 -443.2,E2 -443.2} C_VEL
LIN {X 0,Y 608.437,Z 314.871,A -85,B 0,C 180,E1 -444.198,E2 -444.198} C_VEL
LIN {X 0,Y 608.432,Z 320.946,A -85,B 0,C 180,E1 -445.361,E2 -445.361} C_VEL
LIN {X 0,Y 608.449,Z 324.893,A -85,B 0,C 180,E1 -446.357,E2 -446.357} C_VEL
LIN {X 0,Y 608.425,Z 327.806,A -85,B 0,C 180,E1 -447.351,E2 -447.351} C_VEL
LIN {X 0,Y 608.444,Z 329.2,A -85,B 0,C 180,E1 -448.013,E2 -448.013} C_VEL
LIN {X 0,Y 608.438,Z 330.783,A -85,B 0,C 180,E1 -449.337,E2 -449.337} C_VEL
LIN {X 0,Y 608.434,Z 331,A -85,B 0,C 180,E1 -449.999,E2 -449.999} C_VEL
LIN {X 0,Y 608.448,Z 330.185,A -85,B 0,C 180,E1 -451.323,E2 -451.323} C_VEL
LIN {X 0,Y 608.444,Z 329.203,A -85,B 0,C 180,E1 -451.985,E2 -451.985} C_VEL
LIN {X 0,Y 608.425,Z 327.812,A -85,B 0,C 180,E1 -452.647,E2 -452.647} C_VEL
LIN {X 0,Y 608.449,Z 324.9,A -85,B 0,C 180,E1 -453.641,E2 -453.641} C_VEL
LIN {X 0,Y 608.432,Z 320.955,A -85,B 0,C 180,E1 -454.637,E2 -454.637} C_VEL
LIN {X 0,Y 608.438,Z 314.883,A -85,B 0,C 180,E1 -455.8,E2 -455.8} C_VEL
LIN {X 0,Y 608.461,Z 308.243,A -85,B 0,C 180,E1 -456.798,E2 -456.798} C_VEL
LIN {X 0,Y 608.456,Z 299.999,A -85,B 0,C 180,E1 -457.799,E2 -457.799} C_VEL
LIN {X 0,Y 608.472,Z 291.549,A -85,B 0,C 180,E1 -458.635,E2 -458.635} C_VEL
LIN {X 0,Y 608.48,Z 281.107,A -85,B 0,C 180,E1 -459.472,E2 -459.472} C_VEL
LIN {X 0,Y 608.492,Z 270.776,A -85,B 0,C 180,E1 -460.144,E2 -460.144} C_VEL
LIN {X 0,Y 608.507,Z 259.66,A -85,B 0,C 180,E1 -460.722,E2 -460.722} C_VEL
LIN {X 0,Y 608.52,Z 247.963,A -85,B 0,C 180,E1 -461.19,E2 -461.19} C_VEL
LIN {X 0,Y 608.544,Z 235.319,A -85,B 0,C 180,E1 -461.553,E2 -461.553} C_VEL
LIN {X 0,Y 608.57,Z 221.934,A -85,B 0,C 180,E1 -461.796,E2 -461.796} C_VEL
LIN {X 0,Y 608.451,Z 220.818,A -85,B 0,C 180,E1 -461.83,E2 -461.83} C_VEL
LIN {X 0,Y 608.483,Z 203.591,A -85,B 0,C 180,E1 -464.719,E2 -464.719} C_VEL
LIN {X 0,Y 608.498,Z 186.365,A -85,B 0,C 180,E1 -467.647,E2 -467.647} C_VEL
LIN {X 0,Y 608.491,Z 171.165,A -85,B 0,C 180,E1 -470.272,E2 -470.272} C_VEL
LIN {X 0,Y 608.552,Z 155.966,A -85,B 0,C 180,E1 -472.939,E2 -472.939} C_VEL
LIN {X 0,Y 608.569,Z 140.33,A -85,B 0,C 180,E1 -475.739,E2 -475.739} C_VEL
LIN {X 0,Y 608.436,Z 136.694,A -85,B 0,C 180,E1 -476.449,E2 -476.449} C_VEL
LIN {X 0,Y 608.416,Z 136.703,A -85,B 0,C 180,E1 -479.021,E2 -479.021} C_VEL
LIN {X 0,Y 608.436,Z 136.693,A -85,B 0,C 180,E1 -481.317,E2 -481.317} C_VEL
LIN {X 0,Y 608.466,Z 136.691,A -85,B 0,C 180,E1 -483.734,E2 -483.734} C_VEL
LIN {X 0,Y 608.472,Z 136.691,A -85,B 0,C 180,E1 -486.089,E2 -486.089} C_VEL
LIN {X 0,Y 608.464,Z 136.69,A -85,B 0,C 180,E1 -488.586,E2 -488.586} C_VEL
LIN {X 0,Y 608.427,Z 136.695,A -85,B 0,C 180,E1 -491.338,E2 -491.338} C_VEL
LIN {X 0,Y 608.459,Z 136.696,A -85,B 0,C 180,E1 -494.264,E2 -494.264} C_VEL
LIN {X 0,Y 608.442,Z 136.693,A -85,B 0,C 180,E1 -497.039,E2 -497.039} C_VEL
LIN {X 0,Y 608.441,Z 136.693,A -85,B 0,C 180,E1 -499.696,E2 -499.696} C_VEL
LIN {X 0,Y 608.457,Z 136.693,A -85,B 0,C 180,E1 -502.253,E2 -502.253} C_VEL
LIN {X 0,Y 608.404,Z 136.696,A -85,B 0,C 180,E1 -505.098,E2 -505.098} C_VEL
LIN {X 0,Y 608.464,Z 136.695,A -85,B 0,C 180,E1 -507.474,E2 -507.474} C_VEL
LIN {X 0,Y 608.47,Z 136.688,A -85,B 0,C 180,E1 -510.22,E2 -510.22} C_VEL
LIN {X 0,Y 608.467,Z 136.694,A -85,B 0,C 180,E1 -512.791,E2 -512.791} C_VEL
LIN {X 0,Y 608.436,Z 136.693,A -85,B 0,C 180,E1 -515.428,E2 -515.428} C_VEL
LIN {X 0,Y 608.439,Z 136.692,A -85,B 0,C 180,E1 -518.307,E2 -518.307} C_VEL
LIN {X 0,Y 608.449,Z 136.697,A -85,B 0,C 180,E1 -521.13,E2 -521.13} C_VEL
LIN {X 0,Y 608.461,Z 136.691,A -85,B 0,C 180,E1 -523.906,E2 -523.906} C_VEL
LIN {X 0,Y 608.442,Z 136.692,A -85,B 0,C 180,E1 -526.643,E2 -526.643} C_VEL
LIN {X 0,Y 608.455,Z 136.697,A -85,B 0,C 180,E1 -529.35,E2 -529.35} C_VEL
LIN {X 0,Y 608.448,Z 136.691,A -85,B 0,C 180,E1 -532.033,E2 -532.033} C_VEL
LIN {X 0,Y 608.463,Z 136.693,A -85,B 0,C 180,E1 -534.698,E2 -534.698} C_VEL
LIN {X 0,Y 608.478,Z 136.689,A -85,B 0,C 180,E1 -537.352,E2 -537.352} C_VEL
LIN {X 0,Y 608.446,Z 136.692,A -85,B 0,C 180,E1 -540,E2 -540} C_VEL
LIN {X 0,Y 608.457,Z 136.695,A -85,B 0,C 180,E1 -542.648,E2 -542.648} C_VEL
LIN {X 0,Y 608.445,Z 136.691,A -85,B 0,C 180,E1 -545.302,E2 -545.302} C_VEL
LIN {X 0,Y 608.476,Z 136.694,A -85,B 0,C 180,E1 -547.967,E2 -547.967} C_VEL
LIN {X 0,Y 608.453,Z 136.693,A -85,B 0,C 180,E1 -549.476,E2 -549.476} C_VEL
LIN {X 0,Y 607.77,Z 136.778,A -85,B 0,C 180,E1 -550.029,E2 -550.029} C_VEL
LIN {X 0,Y 604.908,Z 137.135,A -85,B 0,C 180,E1 -550.926,E2 -550.926} C_VEL
LIN {X 0,Y 602.503,Z 137.434,A -85,B 0,C 180,E1 -551.647,E2 -551.647} C_VEL
LIN {X 0,Y 601.476,Z 137.56,A -85,B 0,C 180,E1 -552.204,E2 -552.204} C_VEL
LIN {X 0,Y 601.395,Z 137.571,A -85,B 0,C 180,E1 -552.393,E2 -552.393} C_VEL
LIN {X 0,Y 601.41,Z 137.571,A -85,B 0,C 180,E1 -554.897,E2 -554.897} C_VEL
LIN {X 0,Y 601.415,Z 137.567,A -85,B 0,C 180,E1 -556.986,E2 -556.986} C_VEL
LIN {X 0,Y 601.401,Z 137.574,A -85,B 0,C 180,E1 -559.81,E2 -559.81} C_VEL
LIN {X 0,Y 601.442,Z 137.567,A -85,B 0,C 180,E1 -562.682,E2 -562.682} C_VEL
LIN {X 0,Y 601.386,Z 137.575,A -85,B 0,C 180,E1 -564.879,E2 -564.879} C_VEL
LIN {X 0,Y 601.371,Z 137.573,A -85,B 0,C 180,E1 -567.358,E2 -567.358} C_VEL
LIN {X 0,Y 601.436,Z 137.566,A -85,B 0,C 180,E1 -570.164,E2 -570.164} C_VEL
LIN {X 0,Y 601.41,Z 137.571,A -85,B 0,C 180,E1 -572.717,E2 -572.717} C_VEL
LIN {X 0,Y 601.411,Z 137.57,A -85,B 0,C 180,E1 -575.117,E2 -575.117} C_VEL
LIN {X 0,Y 601.422,Z 137.567,A -85,B 0,C 180,E1 -577.42,E2 -577.42} C_VEL
LIN {X 0,Y 601.39,Z 137.574,A -85,B 0,C 180,E1 -579.997,E2 -579.997} C_VEL
LIN {X 0,Y 601.395,Z 137.571,A -85,B 0,C 180,E1 -582.672,E2 -582.672} C_VEL
LIN {X 0,Y 601.416,Z 137.567,A -85,B 0,C 180,E1 -585.483,E2 -585.483} C_VEL
LIN {X 0,Y 601.415,Z 137.571,A -85,B 0,C 180,E1 -588.408,E2 -588.408} C_VEL
LIN {X 0,Y 601.388,Z 137.571,A -85,B 0,C 180,E1 -590.874,E2 -590.874} C_VEL
LIN {X 0,Y 601.387,Z 137.575,A -85,B 0,C 180,E1 -593.418,E2 -593.418} C_VEL
LIN {X 0,Y 601.425,Z 137.567,A -85,B 0,C 180,E1 -596.066,E2 -596.066} C_VEL
LIN {X 0,Y 601.43,Z 137.565,A -85,B 0,C 180,E1 -599.06,E2 -599.06} C_VEL
LIN {X 0,Y 601.438,Z 137.569,A -85,B 0,C 180,E1 -601.375,E2 -601.375} C_VEL
LIN {X 0,Y 601.388,Z 137.573,A -85,B 0,C 180,E1 -603.637,E2 -603.637} C_VEL
LIN {X 0,Y 601.394,Z 137.57,A -85,B 0,C 180,E1 -605.858,E2 -605.858} C_VEL
LIN {X 0,Y 601.401,Z 137.571,A -85,B 0,C 180,E1 -608.762,E2 -608.762} C_VEL
LIN {X 0,Y 601.417,Z 137.574,A -85,B 0,C 180,E1 -611.609,E2 -611.609} C_VEL
LIN {X 0,Y 601.413,Z 137.568,A -85,B 0,C 180,E1 -614.41,E2 -614.41} C_VEL
LIN {X 0,Y 601.371,Z 137.574,A -85,B 0,C 180,E1 -617.172,E2 -617.172} C_VEL
LIN {X 0,Y 601.426,Z 137.571,A -85,B 0,C 180,E1 -619.906,E2 -619.906} C_VEL
LIN {X 0,Y 601.407,Z 137.568,A -85,B 0,C 180,E1 -622.616,E2 -622.616} C_VEL
LIN {X 0,Y 601.416,Z 137.571,A -85,B 0,C 180,E1 -625.309,E2 -625.309} C_VEL
LIN {X 0,Y 601.434,Z 137.567,A -85,B 0,C 180,E1 -627.992,E2 -627.992} C_VEL
LIN {X 0,Y 601.376,Z 137.573,A -85,B 0,C 180,E1 -630.671,E2 -630.671} C_VEL
LIN {X 0,Y 601.422,Z 137.572,A -85,B 0,C 180,E1 -633.351,E2 -633.351} C_VEL
LIN {X 0,Y 601.416,Z 137.567,A -85,B 0,C 180,E1 -636.038,E2 -636.038} C_VEL
LIN {X 0,Y 601.414,Z 137.571,A -85,B 0,C 180,E1 -638.739,E2 -638.739} C_VEL
LIN {X 0,Y 601.41,Z 137.57,A -85,B 0,C 180,E1 -641.46,E2 -641.46} C_VEL
LIN {X 0,Y 601.38,Z 137.572,A -85,B 0,C 180,E1 -644.207,E2 -644.207} C_VEL
LIN {X 0,Y 601.415,Z 137.574,A -85,B 0,C 180,E1 -646.987,E2 -646.987} C_VEL
LIN {X 0,Y 601.407,Z 137.57,A -85,B 0,C 180,E1 -649.81,E2 -649.81} C_VEL
LIN {X 0,Y 601.406,Z 137.568,A -85,B 0,C 180,E1 -652.684,E2 -652.684} C_VEL
LIN {X 0,Y 601.387,Z 137.573,A -85,B 0,C 180,E1 -654.88,E2 -654.88} C_VEL
LIN {X 0,Y 601.4,Z 137.571,A -85,B 0,C 180,E1 -657.359,E2 -657.359} C_VEL
LIN {X 0,Y 601.395,Z 137.57,A -85,B 0,C 180,E1 -659.395,E2 -659.395} C_VEL
LIN {X 0,Y 601.402,Z 137.572,A -85,B 0,C 180,E1 -661.728,E2 -661.728} C_VEL
LIN {X 0,Y 601.422,Z 137.568,A -85,B 0,C 180,E1 -664.12,E2 -664.12} C_VEL
LIN {X 0,Y 601.405,Z 137.57,A -85,B 0,C 180,E1 -666.584,E2 -666.584} C_VEL
LIN {X 0,Y 601.391,Z 137.57,A -85,B 0,C 180,E1 -669.53,E2 -669.53} C_VEL
LIN {X 0,Y 601.422,Z 137.569,A -85,B 0,C 180,E1 -671.766,E2 -671.766} C_VEL
LIN {X 0,Y 601.402,Z 137.569,A -85,B 0,C 180,E1 -674.533,E2 -674.533} C_VEL
LIN {X 0,Y 601.407,Z 137.571,A -85,B 0,C 180,E1 -677.411,E2 -677.411} C_VEL
LIN {X 0,Y 601.38,Z 137.573,A -85,B 0,C 180,E1 -680.002,E2 -680.002} C_VEL
LIN {X 0,Y 601.399,Z 137.571,A -85,B 0,C 180,E1 -682.623,E2 -682.623} C_VEL
LIN {X 0,Y 601.4,Z 137.571,A -85,B 0,C 180,E1 -685.067,E2 -685.067} C_VEL
LIN {X 0,Y 601.428,Z 137.569,A -85,B 0,C 180,E1 -687.484,E2 -687.484} C_VEL
LIN {X 0,Y 601.435,Z 137.667,A -85,B 0,C 180,E1 -690.089,E2 -690.089} C_VEL
LIN {X 0,Y 601.458,Z 146.489,A -85,B 0,C 180,E1 -692.889,E2 -692.889} C_VEL
LIN {X 0,Y 601.461,Z 156.032,A -85,B 0,C 180,E1 -695.86,E2 -695.86} C_VEL
LIN {X 0,Y 601.371,Z 165.498,A -85,B 0,C 180,E1 -698.759,E2 -698.759} C_VEL
LIN {X 0,Y 601.397,Z 173.557,A -85,B 0,C 180,E1 -701.188,E2 -701.188} C_VEL
LIN {X 0,Y 601.391,Z 183.243,A -85,B 0,C 180,E1 -704.06,E2 -704.06} C_VEL
LIN {X 0,Y 601.386,Z 192.708,A -85,B 0,C 180,E1 -706.828,E2 -706.828} C_VEL
LIN {X 0,Y 601.363,Z 202.173,A -85,B 0,C 180,E1 -709.564,E2 -709.564} C_VEL
LIN {X 0,Y 601.332,Z 210.456,A -85,B 0,C 180,E1 -711.938,E2 -711.938} C_VEL
LIN {X 0,Y 601.36,Z 214.404,A -85,B 0,C 180,E1 -713.065,E2 -713.065} C_VEL
LIN {X 0,Y 601.424,Z 224.551,A -85,B 0,C 180,E1 -713.391,E2 -713.391} C_VEL
LIN {X 0,Y 601.372,Z 232.478,A -85,B 0,C 180,E1 -713.765,E2 -713.765} C_VEL
LIN {X 0,Y 601.344,Z 241.003,A -85,B 0,C 180,E1 -714.299,E2 -714.299} C_VEL
LIN {X 0,Y 601.389,Z 249.033,A -85,B 0,C 180,E1 -714.972,E2 -714.972} C_VEL
LIN {X 0,Y 601.362,Z 255.211,A -85,B 0,C 180,E1 -715.643,E2 -715.643} C_VEL
LIN {X 0,Y 601.374,Z 260.071,A -85,B 0,C 180,E1 -716.315,E2 -716.315} C_VEL
LIN {X 0,Y 601.379,Z 263.821,A -85,B 0,C 180,E1 -716.986,E2 -716.986} C_VEL
LIN {X 0,Y 601.343,Z 267.827,A -85,B 0,C 180,E1 -717.991,E2 -717.991} C_VEL
LIN {X 0,Y 601.348,Z 269.571,A -85,B 0,C 180,E1 -718.661,E2 -718.661} C_VEL
LIN {X 0,Y 601.34,Z 270.616,A -85,B 0,C 180,E1 -719.33,E2 -719.33} C_VEL
LIN {X 0,Y 601.335,Z 270.996,A -85,B 0,C 180,E1 -720,E2 -720} C_VEL
LIN {X 0,Y 601.339,Z 270.714,A -85,B 0,C 180,E1 -720.67,E2 -720.67} C_VEL
LIN {X 0,Y 601.349,Z 269.767,A -85,B 0,C 180,E1 -721.339,E2 -721.339} C_VEL
LIN {X 0,Y 601.342,Z 268.127,A -85,B 0,C 180,E1 -722.009,E2 -722.009} C_VEL
LIN {X 0,Y 601.332,Z 265.743,A -85,B 0,C 180,E1 -722.68,E2 -722.68} C_VEL
LIN {X 0,Y 601.375,Z 260.615,A -85,B 0,C 180,E1 -723.685,E2 -723.685} C_VEL
LIN {X 0,Y 601.378,Z 254.55,A -85,B 0,C 180,E1 -724.524,E2 -724.524} C_VEL
LIN {X 0,Y 601.357,Z 248.242,A -85,B 0,C 180,E1 -725.197,E2 -725.197} C_VEL
LIN {X 0,Y 601.329,Z 241.087,A -85,B 0,C 180,E1 -725.786,E2 -725.786} C_VEL
LIN {X 0,Y 601.352,Z 232.891,A -85,B 0,C 180,E1 -726.302,E2 -726.302} C_VEL
LIN {X 0,Y 601.428,Z 223.075,A -85,B 0,C 180,E1 -726.753,E2 -726.753} C_VEL
LIN {X 0,Y 601.354,Z 214.321,A -85,B 0,C 180,E1 -727.049,E2 -727.049} C_VEL
LIN {X 0,Y 601.319,Z 204.853,A -85,B 0,C 180,E1 -729.757,E2 -729.757} C_VEL
LIN {X 0,Y 601.373,Z 195.384,A -85,B 0,C 180,E1 -732.486,E2 -732.486} C_VEL
LIN {X 0,Y 601.364,Z 185.916,A -85,B 0,C 180,E1 -735.245,E2 -735.245} C_VEL
LIN {X 0,Y 601.393,Z 176.447,A -85,B 0,C 180,E1 -738.04,E2 -738.04} C_VEL
LIN {X 0,Y 601.409,Z 167.271,A -85,B 0,C 180,E1 -740.792,E2 -740.792} C_VEL
LIN {X 0,Y 601.382,Z 158.692,A -85,B 0,C 180,E1 -743.412,E2 -743.412} C_VEL
LIN {X 0,Y 601.431,Z 150.734,A -85,B 0,C 180,E1 -745.87,E2 -745.87} C_VEL
LIN {X 0,Y 601.439,Z 141.704,A -85,B 0,C 180,E1 -748.627,E2 -748.627} C_VEL
LIN {X 0,Y 601.44,Z 137.569,A -85,B 0,C 180,E1 -749.911,E2 -749.911} C_VEL
LIN {X 0,Y 601.422,Z 137.574,A -85,B 0,C 180,E1 -752.715,E2 -752.715} C_VEL
LIN {X 0,Y 601.402,Z 137.575,A -85,B 0,C 180,E1 -755.112,E2 -755.112} C_VEL
LIN {X 0,Y 601.442,Z 137.569,A -85,B 0,C 180,E1 -757.419,E2 -757.419} C_VEL
LIN {X 0,Y 601.408,Z 137.573,A -85,B 0,C 180,E1 -759.995,E2 -759.995} C_VEL
LIN {X 0,Y 601.411,Z 137.574,A -85,B 0,C 180,E1 -762.671,E2 -762.671} C_VEL
LIN {X 0,Y 601.432,Z 137.57,A -85,B 0,C 180,E1 -765.482,E2 -765.482} C_VEL
LIN {X 0,Y 601.424,Z 137.571,A -85,B 0,C 180,E1 -768.407,E2 -768.407} C_VEL
LIN {X 0,Y 601.406,Z 137.573,A -85,B 0,C 180,E1 -770.872,E2 -770.872} C_VEL
LIN {X 0,Y 601.404,Z 137.576,A -85,B 0,C 180,E1 -773.416,E2 -773.416} C_VEL
LIN {X 0,Y 601.422,Z 137.571,A -85,B 0,C 180,E1 -776.066,E2 -776.066} C_VEL
LIN {X 0,Y 601.424,Z 137.572,A -85,B 0,C 180,E1 -778.545,E2 -778.545} C_VEL
LIN {X 0,Y 601.423,Z 137.572,A -85,B 0,C 180,E1 -781.372,E2 -781.372} C_VEL
LIN {X 0,Y 601.432,Z 137.712,A -85,B 0,C 180,E1 -783.45,E2 -783.45} C_VEL
LIN {X 0,Y 601.64,Z 145.819,A -85,B 0,C 180,E1 -784.947,E2 -784.947} C_VEL
LIN {X 0,Y 601.561,Z 161.121,A -85,B 0,C 180,E1 -787.703,E2 -787.703} C_VEL
LIN {X 0,Y 601.516,Z 176.219,A -85,B 0,C 180,E1 -790.371,E2 -790.371} C_VEL
LIN {X 0,Y 601.463,Z 192.765,A -85,B 0,C 180,E1 -793.246,E2 -793.246} C_VEL
LIN {X 0,Y 601.406,Z 208.349,A -85,B 0,C 180,E1 -795.915,E2 -795.915} C_VEL
LIN {X 0,Y 601.409,Z 221.013,A -85,B 0,C 180,E1 -798.049,E2 -798.049} C_VEL
LIN {X 0,Y 601.589,Z 233.4,A -85,B 0,C 180,E1 -798.266,E2 -798.266} C_VEL
LIN {X 0,Y 601.56,Z 247.113,A -85,B 0,C 180,E1 -798.651,E2 -798.651} C_VEL
LIN {X 0,Y 601.538,Z 258.852,A -85,B 0,C 180,E1 -799.115,E2 -799.115} C_VEL
LIN {X 0,Y 601.473,Z 270.742,A -85,B 0,C 180,E1 -799.735,E2 -799.735} C_VEL
LIN {X 0,Y 601.462,Z 282.241,A -85,B 0,C 180,E1 -800.499,E2 -800.499} C_VEL
LIN {X 0,Y 601.436,Z 291.526,A -85,B 0,C 180,E1 -801.261,E2 -801.261} C_VEL
LIN {X 0,Y 601.401,Z 299.981,A -85,B 0,C 180,E1 -802.107,E2 -802.107} C_VEL
LIN {X 0,Y 601.383,Z 308.228,A -85,B 0,C 180,E1 -803.119,E2 -803.119} C_VEL
LIN {X 0,Y 601.372,Z 314.871,A -85,B 0,C 180,E1 -804.13,E2 -804.13} C_VEL
LIN {X 0,Y 601.336,Z 320.946,A -85,B 0,C 180,E1 -805.306,E2 -805.306} C_VEL
LIN {X 0,Y 601.368,Z 324.893,A -85,B 0,C 180,E1 -806.314,E2 -806.314} C_VEL
LIN {X 0,Y 601.325,Z 327.806,A -85,B 0,C 180,E1 -807.319,E2 -807.319} C_VEL
LIN {X 0,Y 601.343,Z 329.2,A -85,B 0,C 180,E1 -807.99,E2 -807.99} C_VEL
LIN {X 0,Y 601.339,Z 330.783,A -85,B 0,C 180,E1 -809.329,E2 -809.329} C_VEL
LIN {X 0,Y 601.335,Z 331,A -85,B 0,C 180,E1 -809.999,E2 -809.999} C_VEL
LIN {X 0,Y 601.347,Z 330.186,A -85,B 0,C 180,E1 -811.338,E2 -811.338} C_VEL
LIN {X 0,Y 601.343,Z 329.204,A -85,B 0,C 180,E1 -812.008,E2 -812.008} C_VEL
LIN {X 0,Y 601.325,Z 327.812,A -85,B 0,C 180,E1 -812.678,E2 -812.678} C_VEL
LIN {X 0,Y 601.368,Z 324.9,A -85,B 0,C 180,E1 -813.684,E2 -813.684} C_VEL
LIN {X 0,Y 601.336,Z 320.955,A -85,B 0,C 180,E1 -814.692,E2 -814.692} C_VEL
LIN {X 0,Y 601.372,Z 314.884,A -85,B 0,C 180,E1 -815.868,E2 -815.868} C_VEL
LIN {X 0,Y 601.387,Z 308.244,A -85,B 0,C 180,E1 -816.879,E2 -816.879} C_VEL
LIN {X 0,Y 601.4,Z 300,A -85,B 0,C 180,E1 -817.891,E2 -817.891} C_VEL
LIN {X 0,Y 601.436,Z 291.55,A -85,B 0,C 180,E1 -818.736,E2 -818.736} C_VEL
LIN {X 0,Y 601.448,Z 281.109,A -85,B 0,C 180,E1 -819.584,E2 -819.584} C_VEL
LIN {X 0,Y 601.472,Z 270.777,A -85,B 0,C 180,E1 -820.263,E2 -820.263} C_VEL
LIN {X 0,Y 601.536,Z 258.874,A -85,B 0,C 180,E1 -820.884,E2 -820.884} C_VEL
LIN {X 0,Y 601.555,Z 246.3,A -85,B 0,C 180,E1 -821.376,E2 -821.376} C_VEL
LIN {X 0,Y 601.589,Z 233.49,A -85,B 0,C 180,E1 -821.731,E2 -821.731} C_VEL
LIN {X 0,Y 601.439,Z 221.177,A -85,B 0,C 180,E1 -821.948,E2 -821.948} C_VEL
LIN {X 0,Y 601.435,Z 205.618,A -85,B 0,C 180,E1 -824.549,E2 -824.549} C_VEL
LIN {X 0,Y 601.493,Z 189.405,A -85,B 0,C 180,E1 -827.333,E2 -827.333} C_VEL
LIN {X 0,Y 601.514,Z 174.205,A -85,B 0,C 180,E1 -829.982,E2 -829.982} C_VEL
LIN {X 0,Y 601.58,Z 159.005,A -85,B 0,C 180,E1 -832.675,E2 -832.675} C_VEL
LIN {X 0,Y 601.652,Z 142.791,A -85,B 0,C 180,E1 -835.606,E2 -835.606} C_VEL
LIN {X 0,Y 601.412,Z 137.57,A -85,B 0,C 180,E1 -836.596,E2 -836.596} C_VEL
LIN {X 0,Y 601.374,Z 137.576,A -85,B 0,C 180,E1 -839.394,E2 -839.394} C_VEL
LIN {X 0,Y 601.394,Z 137.57,A -85,B 0,C 180,E1 -841.726,E2 -841.726} C_VEL
LIN {X 0,Y 601.428,Z 137.573,A -85,B 0,C 180,E1 -844.117,E2 -844.117} C_VEL
LIN {X 0,Y 601.411,Z 137.568,A -85,B 0,C 180,E1 -846.581,E2 -846.581} C_VEL
LIN {X 0,Y 601.409,Z 137.576,A -85,B 0,C 180,E1 -849.125,E2 -849.125} C_VEL
LIN {X 0,Y 601.397,Z 137.569,A -85,B 0,C 180,E1 -851.765,E2 -851.765} C_VEL
LIN {X 0,Y 601.415,Z 137.57,A -85,B 0,C 180,E1 -854.534,E2 -854.534} C_VEL
LIN {X 0,Y 601.405,Z 137.573,A -85,B 0,C 180,E1 -857.329,E2 -857.329} C_VEL
LIN {X 0,Y 601.403,Z 137.569,A -85,B 0,C 180,E1 -860.004,E2 -860.004} C_VEL
LIN {X 0,Y 601.422,Z 137.573,A -85,B 0,C 180,E1 -862.617,E2 -862.617} C_VEL
LIN {X 0,Y 601.37,Z 137.573,A -85,B 0,C 180,E1 -865.065,E2 -865.065} C_VEL
LIN {X 0,Y 601.432,Z 137.571,A -85,B 0,C 180,E1 -867.484,E2 -867.484} C_VEL
LIN {X 0,Y 601.437,Z 137.565,A -85,B 0,C 180,E1 -869.847,E2 -869.847} C_VEL
LIN {X 0,Y 601.409,Z 137.575,A -85,B 0,C 180,E1 -872.635,E2 -872.635} C_VEL
LIN {X 0,Y 601.383,Z 137.571,A -85,B 0,C 180,E1 -875.12,E2 -875.12} C_VEL
LIN {X 0,Y 601.4,Z 137.573,A -85,B 0,C 180,E1 -877.394,E2 -877.394} C_VEL
LIN {X 0,Y 601.393,Z 137.57,A -85,B 0,C 180,E1 -880.19,E2 -880.19} C_VEL
LIN {X 0,Y 601.428,Z 137.569,A -85,B 0,C 180,E1 -883.014,E2 -883.014} C_VEL
LIN {X 0,Y 601.416,Z 137.572,A -85,B 0,C 180,E1 -885.903,E2 -885.903} C_VEL
LIN {X 0,Y 601.391,Z 137.57,A -85,B 0,C 180,E1 -888.541,E2 -888.541} C_VEL
LIN {X 0,Y 601.423,Z 137.571,A -85,B 0,C 180,E1 -891.262,E2 -891.262} C_VEL
LIN {X 0,Y 601.398,Z 137.571,A -85,B 0,C 180,E1 -893.963,E2 -893.963} C_VEL
LIN {X 0,Y 601.421,Z 137.568,A -85,B 0,C 180,E1 -896.65,E2 -896.65} C_VEL
LIN {X 0,Y 601.453,Z 137.568,A -85,B 0,C 180,E1 -899.33,E2 -899.33} C_VEL
LIN {X 0,Y 601.379,Z 137.571,A -85,B 0,C 180,E1 -902.009,E2 -902.009} C_VEL
LIN {X 0,Y 601.428,Z 137.571,A -85,B 0,C 180,E1 -904.692,E2 -904.692} C_VEL
LIN {X 0,Y 601.441,Z 137.565,A -85,B 0,C 180,E1 -907.385,E2 -907.385} C_VEL
LIN {X 0,Y 601.426,Z 137.567,A -85,B 0,C 180,E1 -910.095,E2 -910.095} C_VEL
LIN {X 0,Y 601.395,Z 137.571,A -85,B 0,C 180,E1 -912.393,E2 -912.393} C_VEL
LIN {X 0,Y 600.735,Z 137.659,A -85,B 0,C 180,E1 -912.952,E2 -912.952} C_VEL
LIN {X 0,Y 597.883,Z 138.012,A -85,B 0,C 180,E1 -913.86,E2 -913.86} C_VEL
LIN {X 0,Y 595.465,Z 138.316,A -85,B 0,C 180,E1 -914.59,E2 -914.59} C_VEL
LIN {X 0,Y 594.423,Z 138.439,A -85,B 0,C 180,E1 -915.153,E2 -915.153} C_VEL
LIN {X 0,Y 594.336,Z 138.449,A -85,B 0,C 180,E1 -915.344,E2 -915.344} C_VEL
LIN {X 0,Y 594.368,Z 138.452,A -85,B 0,C 180,E1 -917.905,E2 -917.905} C_VEL
LIN {X 0,Y 594.373,Z 138.447,A -85,B 0,C 180,E1 -920.919,E2 -920.919} C_VEL
LIN {X 0,Y 594.383,Z 138.443,A -85,B 0,C 180,E1 -923.704,E2 -923.704} C_VEL
LIN {X 0,Y 594.343,Z 138.451,A -85,B 0,C 180,E1 -926.702,E2 -926.702} C_VEL
LIN {X 0,Y 594.36,Z 138.446,A -85,B 0,C 180,E1 -929,E2 -929} C_VEL
LIN {X 0,Y 594.382,Z 138.447,A -85,B 0,C 180,E1 -931.646,E2 -931.646} C_VEL
LIN {X 0,Y 594.392,Z 138.447,A -85,B 0,C 180,E1 -934.579,E2 -934.579} C_VEL
LIN {X 0,Y 594.371,Z 138.445,A -85,B 0,C 180,E1 -937.088,E2 -937.088} C_VEL
LIN {X 0,Y 594.348,Z 138.455,A -85,B 0,C 180,E1 -939.774,E2 -939.774} C_VEL
LIN {X 0,Y 594.35,Z 138.447,A -85,B 0,C 180,E1 -942.377,E2 -942.377} C_VEL
LIN {X 0,Y 594.354,Z 138.449,A -85,B 0,C 180,E1 -945.192,E2 -945.192} C_VEL
LIN {X 0,Y 594.365,Z 138.447,A -85,B 0,C 180,E1 -947.626,E2 -947.626} C_VEL
LIN {X 0,Y 594.36,Z 138.447,A -85,B 0,C 180,E1 -950.32,E2 -950.32} C_VEL
LIN {X 0,Y 594.368,Z 138.448,A -85,B 0,C 180,E1 -952.914,E2 -952.914} C_VEL
LIN {X 0,Y 594.375,Z 138.444,A -85,B 0,C 180,E1 -955.863,E2 -955.863} C_VEL
LIN {X 0,Y 594.387,Z 138.445,A -85,B 0,C 180,E1 -958.652,E2 -958.652} C_VEL
LIN {X 0,Y 594.383,Z 138.444,A -85,B 0,C 180,E1 -961.043,E2 -961.043} C_VEL
LIN {X 0,Y 594.378,Z 138.451,A -85,B 0,C 180,E1 -963.302,E2 -963.302} C_VEL
LIN {X 0,Y 594.343,Z 138.451,A -85,B 0,C 180,E1 -966.295,E2 -966.295} C_VEL
LIN {X 0,Y 594.391,Z 138.442,A -85,B 0,C 180,E1 -969.225,E2 -969.225} C_VEL
LIN {X 0,Y 594.353,Z 138.449,A -85,B 0,C 180,E1 -972.096,E2 -972.096} C_VEL
LIN {X 0,Y 594.364,Z 138.446,A -85,B 0,C 180,E1 -974.22,E2 -974.22} C_VEL
LIN {X 0,Y 594.366,Z 138.448,A -85,B 0,C 180,E1 -976.322,E2 -976.322} C_VEL
LIN {X 0,Y 594.346,Z 138.448,A -85,B 0,C 180,E1 -979.095,E2 -979.095} C_VEL
LIN {X 0,Y 594.413,Z 138.445,A -85,B 0,C 180,E1 -981.844,E2 -981.844} C_VEL
LIN {X 0,Y 594.393,Z 138.443,A -85,B 0,C 180,E1 -984.573,E2 -984.573} C_VEL
LIN {X 0,Y 594.393,Z 138.443,A -85,B 0,C 180,E1 -987.29,E2 -987.29} C_VEL
LIN {X 0,Y 594.413,Z 138.445,A -85,B 0,C 180,E1 -990.001,E2 -990.001} C_VEL
LIN {X 0,Y 594.381,Z 138.443,A -85,B 0,C 180,E1 -992.712,E2 -992.712} C_VEL
LIN {X 0,Y 594.398,Z 138.445,A -85,B 0,C 180,E1 -995.429,E2 -995.429} C_VEL
LIN {X 0,Y 594.416,Z 138.442,A -85,B 0,C 180,E1 -998.158,E2 -998.158} C_VEL
LIN {X 0,Y 594.379,Z 138.444,A -85,B 0,C 180,E1 -1001.067,E2 -1001.067} C_VEL
LIN {X 0,Y 594.352,Z 138.452,A -85,B 0,C 180,E1 -1003.681,E2 -1003.681} C_VEL
LIN {X 0,Y 594.367,Z 138.45,A -85,B 0,C 180,E1 -1006.71,E2 -1006.71} C_VEL
LIN {X 0,Y 594.372,Z 138.445,A -85,B 0,C 180,E1 -1009.335,E2 -1009.335} C_VEL
LIN {X 0,Y 594.364,Z 138.447,A -85,B 0,C 180,E1 -1011.504,E2 -1011.504} C_VEL
LIN {X 0,Y 594.347,Z 138.448,A -85,B 0,C 180,E1 -1014.449,E2 -1014.449} C_VEL
LIN {X 0,Y 594.37,Z 138.448,A -85,B 0,C 180,E1 -1016.701,E2 -1016.701} C_VEL
LIN {X 0,Y 594.36,Z 138.447,A -85,B 0,C 180,E1 -1019.778,E2 -1019.778} C_VEL
LIN {X 0,Y 594.365,Z 138.451,A -85,B 0,C 180,E1 -1022.148,E2 -1022.148} C_VEL
LIN {X 0,Y 594.384,Z 138.443,A -85,B 0,C 180,E1 -1024.581,E2 -1024.581} C_VEL
LIN {X 0,Y 594.357,Z 138.447,A -85,B 0,C 180,E1 -1027.604,E2 -1027.604} C_VEL
LIN {X 0,Y 594.358,Z 138.451,A -85,B 0,C 180,E1 -1030.569,E2 -1030.569} C_VEL
LIN {X 0,Y 594.369,Z 138.447,A -85,B 0,C 180,E1 -1033.3,E2 -1033.3} C_VEL
LIN {X 0,Y 594.365,Z 138.446,A -85,B 0,C 180,E1 -1036.162,E2 -1036.162} C_VEL
LIN {X 0,Y 594.38,Z 138.447,A -85,B 0,C 180,E1 -1038.536,E2 -1038.536} C_VEL
LIN {X 0,Y 594.358,Z 138.446,A -85,B 0,C 180,E1 -1041.3,E2 -1041.3} C_VEL
LIN {X 0,Y 594.348,Z 138.454,A -85,B 0,C 180,E1 -1043.755,E2 -1043.755} C_VEL
LIN {X 0,Y 594.368,Z 138.445,A -85,B 0,C 180,E1 -1046.238,E2 -1046.238} C_VEL
LIN {X 0,Y 594.374,Z 138.449,A -85,B 0,C 180,E1 -1048.65,E2 -1048.65} C_VEL
LIN {X 0,Y 594.422,Z 138.556,A -85,B 0,C 180,E1 -1050.007,E2 -1050.007} C_VEL
LIN {X 0,Y 594.435,Z 146.449,A -85,B 0,C 180,E1 -1052.542,E2 -1052.542} C_VEL
LIN {X 0,Y 594.363,Z 154.821,A -85,B 0,C 180,E1 -1055.18,E2 -1055.18} C_VEL
LIN {X 0,Y 594.35,Z 163.134,A -85,B 0,C 180,E1 -1057.766,E2 -1057.766} C_VEL
LIN {X 0,Y 594.322,Z 171.415,A -85,B 0,C 180,E1 -1060.305,E2 -1060.305} C_VEL
LIN {X 0,Y 594.312,Z 179.696,A -85,B 0,C 180,E1 -1062.804,E2 -1062.804} C_VEL
LIN {X 0,Y 594.312,Z 189.161,A -85,B 0,C 180,E1 -1065.621,E2 -1065.621} C_VEL
LIN {X 0,Y 594.276,Z 198.626,A -85,B 0,C 180,E1 -1068.402,E2 -1068.402} C_VEL
LIN {X 0,Y 594.294,Z 209.274,A -85,B 0,C 180,E1 -1071.499,E2 -1071.499} C_VEL
LIN {X 0,Y 594.263,Z 214.377,A -85,B 0,C 180,E1 -1072.973,E2 -1072.973} C_VEL
LIN {X 0,Y 594.391,Z 224.729,A -85,B 0,C 180,E1 -1073.319,E2 -1073.319} C_VEL
LIN {X 0,Y 594.311,Z 232.915,A -85,B 0,C 180,E1 -1073.715,E2 -1073.715} C_VEL
LIN {X 0,Y 594.27,Z 241.013,A -85,B 0,C 180,E1 -1074.231,E2 -1074.231} C_VEL
LIN {X 0,Y 594.327,Z 249.038,A -85,B 0,C 180,E1 -1074.912,E2 -1074.912} C_VEL
LIN {X 0,Y 594.286,Z 255.214,A -85,B 0,C 180,E1 -1075.591,E2 -1075.591} C_VEL
LIN {X 0,Y 594.3,Z 260.074,A -85,B 0,C 180,E1 -1076.271,E2 -1076.271} C_VEL
LIN {X 0,Y 594.279,Z 263.824,A -85,B 0,C 180,E1 -1076.949,E2 -1076.949} C_VEL
LIN {X 0,Y 594.244,Z 267.83,A -85,B 0,C 180,E1 -1077.967,E2 -1077.967} C_VEL
LIN {X 0,Y 594.248,Z 269.572,A -85,B 0,C 180,E1 -1078.645,E2 -1078.645} C_VEL
LIN {X 0,Y 594.24,Z 270.617,A -85,B 0,C 180,E1 -1079.322,E2 -1079.322} C_VEL
LIN {X 0,Y 594.236,Z 270.996,A -85,B 0,C 180,E1 -1080,E2 -1080} C_VEL
LIN {X 0,Y 594.239,Z 270.713,A -85,B 0,C 180,E1 -1080.678,E2 -1080.678} C_VEL
LIN {X 0,Y 594.249,Z 269.766,A -85,B 0,C 180,E1 -1081.355,E2 -1081.355} C_VEL
LIN {X 0,Y 594.242,Z 268.125,A -85,B 0,C 180,E1 -1082.033,E2 -1082.033} C_VEL
LIN {X 0,Y 594.237,Z 265.741,A -85,B 0,C 180,E1 -1082.712,E2 -1082.712} C_VEL
LIN {X 0,Y 594.3,Z 260.612,A -85,B 0,C 180,E1 -1083.729,E2 -1083.729} C_VEL
LIN {X 0,Y 594.31,Z 254.546,A -85,B 0,C 180,E1 -1084.578,E2 -1084.578} C_VEL
LIN {X 0,Y 594.282,Z 248.236,A -85,B 0,C 180,E1 -1085.259,E2 -1085.259} C_VEL
LIN {X 0,Y 594.271,Z 241.081,A -85,B 0,C 180,E1 -1085.855,E2 -1085.855} C_VEL
LIN {X 0,Y 594.299,Z 232.827,A -85,B 0,C 180,E1 -1086.38,E2 -1086.38} C_VEL
LIN {X 0,Y 594.399,Z 223.062,A -85,B 0,C 180,E1 -1086.833,E2 -1086.833} C_VEL
LIN {X 0,Y 594.267,Z 214.393,A -85,B 0,C 180,E1 -1087.112,E2 -1087.112} C_VEL
LIN {X 0,Y 594.242,Z 206.034,A -85,B 0,C 180,E1 -1089.531,E2 -1089.531} C_VEL
LIN {X 0,Y 594.298,Z 196.566,A -85,B 0,C 180,E1 -1092.29,E2 -1092.29} C_VEL
LIN {X 0,Y 594.294,Z 187.098,A -85,B 0,C 180,E1 -1095.08,E2 -1095.08} C_VEL
LIN {X 0,Y 594.314,Z 178.812,A -85,B 0,C 180,E1 -1097.551,E2 -1097.551} C_VEL
LIN {X 0,Y 594.379,Z 169.343,A -85,B 0,C 180,E1 -1100.415,E2 -1100.415} C_VEL
LIN {X 0,Y 594.338,Z 159.851,A -85,B 0,C 180,E1 -1103.337,E2 -1103.337} C_VEL
LIN {X 0,Y 594.404,Z 151.225,A -85,B 0,C 180,E1 -1106.025,E2 -1106.025} C_VEL
LIN {X 0,Y 594.416,Z 142.824,A -85,B 0,C 180,E1 -1108.595,E2 -1108.595} C_VEL
LIN {X 0,Y 594.402,Z 138.447,A -85,B 0,C 180,E1 -1109.95,E2 -1109.95} C_VEL
LIN {X 0,Y 594.381,Z 138.449,A -85,B 0,C 180,E1 -1112.95,E2 -1112.95} C_VEL
LIN {X 0,Y 594.356,Z 138.451,A -85,B 0,C 180,E1 -1115.409,E2 -1115.409} C_VEL
LIN {X 0,Y 594.392,Z 138.448,A -85,B 0,C 180,E1 -1117.94,E2 -1117.94} C_VEL
LIN {X 0,Y 594.377,Z 138.448,A -85,B 0,C 180,E1 -1120.821,E2 -1120.821} C_VEL
LIN {X 0,Y 594.37,Z 138.45,A -85,B 0,C 180,E1 -1123.299,E2 -1123.299} C_VEL
LIN {X 0,Y 594.374,Z 138.449,A -85,B 0,C 180,E1 -1126.16,E2 -1126.16} C_VEL
LIN {X 0,Y 594.382,Z 138.448,A -85,B 0,C 180,E1 -1128.535,E2 -1128.535} C_VEL
LIN {X 0,Y 594.376,Z 138.451,A -85,B 0,C 180,E1 -1131.297,E2 -1131.297} C_VEL
LIN {X 0,Y 594.355,Z 138.452,A -85,B 0,C 180,E1 -1133.755,E2 -1133.755} C_VEL
LIN {X 0,Y 594.37,Z 138.45,A -85,B 0,C 180,E1 -1136.237,E2 -1136.237} C_VEL
LIN {X 0,Y 594.375,Z 138.451,A -85,B 0,C 180,E1 -1138.649,E2 -1138.649} C_VEL
LIN {X 0,Y 594.382,Z 138.452,A -85,B 0,C 180,E1 -1141.043,E2 -1141.043} C_VEL
LIN {X 0,Y 594.407,Z 138.544,A -85,B 0,C 180,E1 -1143.23,E2 -1143.23} C_VEL
LIN {X 0,Y 594.755,Z 142.903,A -85,B 0,C 180,E1 -1144.073,E2 -1144.073} C_VEL
LIN {X 0,Y 594.636,Z 157.979,A -85,B 0,C 180,E1 -1146.859,E2 -1146.859} C_VEL
LIN {X 0,Y 594.532,Z 173.179,A -85,B 0,C 180,E1 -1149.59,E2 -1149.59} C_VEL
LIN {X 0,Y 594.501,Z 188.379,A -85,B 0,C 180,E1 -1152.277,E2 -1152.277} C_VEL
LIN {X 0,Y 594.409,Z 204.592,A -85,B 0,C 180,E1 -1155.097,E2 -1155.097} C_VEL
LIN {X 0,Y 594.393,Z 221.013,A -85,B 0,C 180,E1 -1157.906,E2 -1157.906} C_VEL
LIN {X 0,Y 594.69,Z 228.039,A -85,B 0,C 180,E1 -1158.02,E2 -1158.02} C_VEL
LIN {X 0,Y 594.634,Z 240.945,A -85,B 0,C 180,E1 -1158.322,E2 -1158.322} C_VEL
LIN {X 0,Y 594.581,Z 253.423,A -85,B 0,C 180,E1 -1158.751,E2 -1158.751} C_VEL
LIN {X 0,Y 594.546,Z 264.614,A -85,B 0,C 180,E1 -1159.269,E2 -1159.269} C_VEL
LIN {X 0,Y 594.467,Z 276.186,A -85,B 0,C 180,E1 -1159.956,E2 -1159.956} C_VEL
LIN {X 0,Y 594.415,Z 286.585,A -85,B 0,C 180,E1 -1160.729,E2 -1160.729} C_VEL
LIN {X 0,Y 594.366,Z 295.102,A -85,B 0,C 180,E1 -1161.499,E2 -1161.499} C_VEL
LIN {X 0,Y 594.348,Z 302.952,A -85,B 0,C 180,E1 -1162.354,E2 -1162.354} C_VEL
LIN {X 0,Y 594.283,Z 310.809,A -85,B 0,C 180,E1 -1163.408,E2 -1163.408} C_VEL
LIN {X 0,Y 594.289,Z 317.675,A -85,B 0,C 180,E1 -1164.57,E2 -1164.57} C_VEL
LIN {X 0,Y 594.27,Z 322.367,A -85,B 0,C 180,E1 -1165.59,E2 -1165.59} C_VEL
LIN {X 0,Y 594.267,Z 325.953,A -85,B 0,C 180,E1 -1166.609,E2 -1166.609} C_VEL
LIN {X 0,Y 594.226,Z 327.806,A -85,B 0,C 180,E1 -1167.287,E2 -1167.287} C_VEL
LIN {X 0,Y 594.242,Z 329.199,A -85,B 0,C 180,E1 -1167.966,E2 -1167.966} C_VEL
LIN {X 0,Y 594.239,Z 330.783,A -85,B 0,C 180,E1 -1169.321,E2 -1169.321} C_VEL
LIN {X 0,Y 594.236,Z 331,A -85,B 0,C 180,E1 -1169.999,E2 -1169.999} C_VEL
LIN {X 0,Y 594.247,Z 330.186,A -85,B 0,C 180,E1 -1171.354,E2 -1171.354} C_VEL
LIN {X 0,Y 594.242,Z 329.203,A -85,B 0,C 180,E1 -1172.032,E2 -1172.032} C_VEL
LIN {X 0,Y 594.226,Z 327.812,A -85,B 0,C 180,E1 -1172.71,E2 -1172.71} C_VEL
LIN {X 0,Y 594.289,Z 324.9,A -85,B 0,C 180,E1 -1173.728,E2 -1173.728} C_VEL
LIN {X 0,Y 594.241,Z 320.954,A -85,B 0,C 180,E1 -1174.748,E2 -1174.748} C_VEL
LIN {X 0,Y 594.305,Z 314.885,A -85,B 0,C 180,E1 -1175.938,E2 -1175.938} C_VEL
LIN {X 0,Y 594.311,Z 308.245,A -85,B 0,C 180,E1 -1176.961,E2 -1176.961} C_VEL
LIN {X 0,Y 594.359,Z 300,A -85,B 0,C 180,E1 -1177.985,E2 -1177.985} C_VEL
LIN {X 0,Y 594.382,Z 291.55,A -85,B 0,C 180,E1 -1178.841,E2 -1178.841} C_VEL
LIN {X 0,Y 594.429,Z 281.11,A -85,B 0,C 180,E1 -1179.698,E2 -1179.698} C_VEL
LIN {X 0,Y 594.482,Z 270.779,A -85,B 0,C 180,E1 -1180.385,E2 -1180.385} C_VEL
LIN {X 0,Y 594.534,Z 258.577,A -85,B 0,C 180,E1 -1181.027,E2 -1181.027} C_VEL
LIN {X 0,Y 594.581,Z 246.49,A -85,B 0,C 180,E1 -1181.505,E2 -1181.505} C_VEL
LIN {X 0,Y 594.64,Z 233.489,A -85,B 0,C 180,E1 -1181.871,E2 -1181.871} C_VEL
LIN {X 0,Y 594.545,Z 222.217,A -85,B 0,C 180,E1 -1182.074,E2 -1182.074} C_VEL
LIN {X 0,Y 594.365,Z 220.818,A -85,B 0,C 180,E1 -1182.114,E2 -1182.114} C_VEL
LIN {X 0,Y 594.407,Z 204.605,A -85,B 0,C 180,E1 -1184.9,E2 -1184.9} C_VEL
LIN {X 0,Y 594.499,Z 188.391,A -85,B 0,C 180,E1 -1187.721,E2 -1187.721} C_VEL
LIN {X 0,Y 594.531,Z 173.191,A -85,B 0,C 180,E1 -1190.408,E2 -1190.408} C_VEL
LIN {X 0,Y 594.633,Z 157.991,A -85,B 0,C 180,E1 -1193.139,E2 -1193.139} C_VEL
LIN {X 0,Y 594.712,Z 142.809,A -85,B 0,C 180,E1 -1195.927,E2 -1195.927} C_VEL
LIN {X 0,Y 594.395,Z 138.445,A -85,B 0,C 180,E1 -1196.769,E2 -1196.769} C_VEL
LIN {X 0,Y 594.34,Z 138.449,A -85,B 0,C 180,E1 -1199.777,E2 -1199.777} C_VEL
LIN {X 0,Y 594.366,Z 138.449,A -85,B 0,C 180,E1 -1202.145,E2 -1202.145} C_VEL
LIN {X 0,Y 594.396,Z 138.443,A -85,B 0,C 180,E1 -1204.577,E2 -1204.577} C_VEL
LIN {X 0,Y 594.382,Z 138.446,A -85,B 0,C 180,E1 -1207.085,E2 -1207.085} C_VEL
LIN {X 0,Y 594.347,Z 138.448,A -85,B 0,C 180,E1 -1209.771,E2 -1209.771} C_VEL
LIN {X 0,Y 594.352,Z 138.453,A -85,B 0,C 180,E1 -1212.375,E2 -1212.375} C_VEL
LIN {X 0,Y 594.354,Z 138.447,A -85,B 0,C 180,E1 -1215.19,E2 -1215.19} C_VEL
LIN {X 0,Y 594.364,Z 138.452,A -85,B 0,C 180,E1 -1217.624,E2 -1217.624} C_VEL
LIN {X 0,Y 594.387,Z 138.444,A -85,B 0,C 180,E1 -1220.32,E2 -1220.32} C_VEL
LIN {X 0,Y 594.365,Z 138.448,A -85,B 0,C 180,E1 -1222.912,E2 -1222.912} C_VEL
LIN {X 0,Y 594.365,Z 138.448,A -85,B 0,C 180,E1 -1226.238,E2 -1226.238} C_VEL
LIN {X 0,Y 594.38,Z 138.444,A -85,B 0,C 180,E1 -1228.65,E2 -1228.65} C_VEL
LIN {X 0,Y 594.375,Z 138.451,A -85,B 0,C 180,E1 -1231.04,E2 -1231.04} C_VEL
LIN {X 0,Y 594.385,Z 138.446,A -85,B 0,C 180,E1 -1233.974,E2 -1233.974} C_VEL
LIN {X 0,Y 594.365,Z 138.448,A -85,B 0,C 180,E1 -1236.295,E2 -1236.295} C_VEL
LIN {X 0,Y 594.398,Z 138.447,A -85,B 0,C 180,E1 -1239.224,E2 -1239.224} C_VEL
LIN {X 0,Y 594.375,Z 138.445,A -85,B 0,C 180,E1 -1242.096,E2 -1242.096} C_VEL
LIN {X 0,Y 594.363,Z 138.451,A -85,B 0,C 180,E1 -1244.219,E2 -1244.219} C_VEL
LIN {X 0,Y 594.368,Z 138.449,A -85,B 0,C 180,E1 -1246.321,E2 -1246.321} C_VEL
LIN {X 0,Y 594.364,Z 138.448,A -85,B 0,C 180,E1 -1249.094,E2 -1249.094} C_VEL
LIN {X 0,Y 594.366,Z 138.445,A -85,B 0,C 180,E1 -1251.843,E2 -1251.843} C_VEL
LIN {X 0,Y 594.387,Z 138.449,A -85,B 0,C 180,E1 -1254.572,E2 -1254.572} C_VEL
LIN {X 0,Y 594.406,Z 138.442,A -85,B 0,C 180,E1 -1257.289,E2 -1257.289} C_VEL
LIN {X 0,Y 594.386,Z 138.444,A -85,B 0,C 180,E1 -1260,E2 -1260} C_VEL
LIN {X 0,Y 594.388,Z 138.448,A -85,B 0,C 180,E1 -1262.711,E2 -1262.711} C_VEL
LIN {X 0,Y 594.374,Z 138.444,A -85,B 0,C 180,E1 -1265.428,E2 -1265.428} C_VEL
LIN {X 0,Y 594.412,Z 138.443,A -85,B 0,C 180,E1 -1268.157,E2 -1268.157} C_VEL
LIN {X 0,Y 594.385,Z 138.448,A -85,B 0,C 180,E1 -1271.08,E2 -1271.08} C_VEL
LIN {X 0,Y 594.352,Z 138.447,A -85,B 0,C 180,E1 -1273.68,E2 -1273.68} C_VEL
LIN {X 0,Y 594.336,Z 138.449,A -85,B 0,C 180,E1 -1275.344,E2 -1275.344} C_VEL
LIN {X 0,Y 593.666,Z 138.536,A -85,B 0,C 180,E1 -1275.91,E2 -1275.91} C_VEL
LIN {X 0,Y 590.817,Z 138.892,A -85,B 0,C 180,E1 -1276.828,E2 -1276.828} C_VEL
LIN {X 0,Y 588.418,Z 139.193,A -85,B 0,C 180,E1 -1277.567,E2 -1277.567} C_VEL
LIN {X 0,Y 587.394,Z 139.319,A -85,B 0,C 180,E1 -1278.138,E2 -1278.138} C_VEL
LIN {X 0,Y 587.313,Z 139.326,A -85,B 0,C 180,E1 -1278.331,E2 -1278.331} C_VEL
LIN {X 0,Y 587.344,Z 139.324,A -85,B 0,C 180,E1 -1281.045,E2 -1281.045} C_VEL
LIN {X 0,Y 587.354,Z 139.322,A -85,B 0,C 180,E1 -1283.257,E2 -1283.257} C_VEL
LIN {X 0,Y 587.322,Z 139.328,A -85,B 0,C 180,E1 -1286.177,E2 -1286.177} C_VEL
LIN {X 0,Y 587.333,Z 139.324,A -85,B 0,C 180,E1 -1289.38,E2 -1289.38} C_VEL
LIN {X 0,Y 587.344,Z 139.322,A -85,B 0,C 180,E1 -1291.839,E2 -1291.839} C_VEL
LIN {X 0,Y 587.351,Z 139.322,A -85,B 0,C 180,E1 -1294.351,E2 -1294.351} C_VEL
LIN {X 0,Y 587.34,Z 139.323,A -85,B 0,C 180,E1 -1296.748,E2 -1296.748} C_VEL
LIN {X 0,Y 587.318,Z 139.325,A -85,B 0,C 180,E1 -1299.362,E2 -1299.362} C_VEL
LIN {X 0,Y 587.324,Z 139.323,A -85,B 0,C 180,E1 -1302.109,E2 -1302.109} C_VEL
LIN {X 0,Y 587.307,Z 139.328,A -85,B 0,C 180,E1 -1305.09,E2 -1305.09} C_VEL
LIN {X 0,Y 587.344,Z 139.324,A -85,B 0,C 180,E1 -1307.929,E2 -1307.929} C_VEL
LIN {X 0,Y 587.317,Z 139.323,A -85,B 0,C 180,E1 -1310.64,E2 -1310.64} C_VEL
LIN {X 0,Y 587.309,Z 139.33,A -85,B 0,C 180,E1 -1313.298,E2 -1313.298} C_VEL
LIN {X 0,Y 587.356,Z 139.319,A -85,B 0,C 180,E1 -1315.781,E2 -1315.781} C_VEL
LIN {X 0,Y 587.346,Z 139.327,A -85,B 0,C 180,E1 -1318.233,E2 -1318.233} C_VEL
LIN {X 0,Y 587.349,Z 139.32,A -85,B 0,C 180,E1 -1320.867,E2 -1320.867} C_VEL
LIN {X 0,Y 587.327,Z 139.324,A -85,B 0,C 180,E1 -1323.722,E2 -1323.722} C_VEL
LIN {X 0,Y 587.296,Z 139.332,A -85,B 0,C 180,E1 -1326.742,E2 -1326.742} C_VEL
LIN {X 0,Y 587.321,Z 139.326,A -85,B 0,C 180,E1 -1329.696,E2 -1329.696} C_VEL
LIN {X 0,Y 587.351,Z 139.319,A -85,B 0,C 180,E1 -1332.595,E2 -1332.595} C_VEL
LIN {X 0,Y 587.33,Z 139.324,A -85,B 0,C 180,E1 -1335.448,E2 -1335.448} C_VEL
LIN {X 0,Y 587.316,Z 139.329,A -85,B 0,C 180,E1 -1338.264,E2 -1338.264} C_VEL
LIN {X 0,Y 587.317,Z 139.324,A -85,B 0,C 180,E1 -1341.052,E2 -1341.052} C_VEL
LIN {X 0,Y 587.376,Z 139.322,A -85,B 0,C 180,E1 -1343.267,E2 -1343.267} C_VEL
LIN {X 0,Y 587.315,Z 139.324,A -85,B 0,C 180,E1 -1345.884,E2 -1345.884} C_VEL
LIN {X 0,Y 587.372,Z 139.318,A -85,B 0,C 180,E1 -1347.944,E2 -1347.944} C_VEL
LIN {X 0,Y 587.382,Z 139.321,A -85,B 0,C 180,E1 -1350.001,E2 -1350.001} C_VEL
LIN {X 0,Y 587.351,Z 139.319,A -85,B 0,C 180,E1 -1352.744,E2 -1352.744} C_VEL
LIN {X 0,Y 587.362,Z 139.321,A -85,B 0,C 180,E1 -1355.494,E2 -1355.494} C_VEL
LIN {X 0,Y 587.368,Z 139.321,A -85,B 0,C 180,E1 -1358.256,E2 -1358.256} C_VEL
LIN {X 0,Y 587.353,Z 139.319,A -85,B 0,C 180,E1 -1361.135,E2 -1361.135} C_VEL
LIN {X 0,Y 587.304,Z 139.325,A -85,B 0,C 180,E1 -1364.236,E2 -1364.236} C_VEL
LIN {X 0,Y 587.337,Z 139.327,A -85,B 0,C 180,E1 -1366.81,E2 -1366.81} C_VEL
LIN {X 0,Y 587.318,Z 139.324,A -85,B 0,C 180,E1 -1369.577,E2 -1369.577} C_VEL
LIN {X 0,Y 587.318,Z 139.329,A -85,B 0,C 180,E1 -1371.775,E2 -1371.775} C_VEL
LIN {X 0,Y 587.301,Z 139.326,A -85,B 0,C 180,E1 -1374.762,E2 -1374.762} C_VEL
LIN {X 0,Y 587.302,Z 139.325,A -85,B 0,C 180,E1 -1377.683,E2 -1377.683} C_VEL
LIN {X 0,Y 587.321,Z 139.328,A -85,B 0,C 180,E1 -1380.172,E2 -1380.172} C_VEL
LIN {X 0,Y 587.34,Z 139.322,A -85,B 0,C 180,E1 -1382.58,E2 -1382.58} C_VEL
LIN {X 0,Y 587.329,Z 139.325,A -85,B 0,C 180,E1 -1385.056,E2 -1385.056} C_VEL
LIN {X 0,Y 587.289,Z 139.327,A -85,B 0,C 180,E1 -1387.832,E2 -1387.832} C_VEL
LIN {X 0,Y 587.304,Z 139.33,A -85,B 0,C 180,E1 -1390.256,E2 -1390.256} C_VEL
LIN {X 0,Y 587.318,Z 139.324,A -85,B 0,C 180,E1 -1393.118,E2 -1393.118} C_VEL
LIN {X 0,Y 587.317,Z 139.324,A -85,B 0,C 180,E1 -1396.049,E2 -1396.049} C_VEL
LIN {X 0,Y 587.337,Z 139.326,A -85,B 0,C 180,E1 -1398.926,E2 -1398.926} C_VEL
LIN {X 0,Y 587.305,Z 139.325,A -85,B 0,C 180,E1 -1401.519,E2 -1401.519} C_VEL
LIN {X 0,Y 587.297,Z 139.326,A -85,B 0,C 180,E1 -1404.463,E2 -1404.463} C_VEL
LIN {X 0,Y 587.34,Z 139.324,A -85,B 0,C 180,E1 -1406.889,E2 -1406.889} C_VEL
LIN {X 0,Y 587.365,Z 139.322,A -85,B 0,C 180,E1 -1409.881,E2 -1409.881} C_VEL
LIN {X 0,Y 587.431,Z 146.746,A -85,B 0,C 180,E1 -1412.293,E2 -1412.293} C_VEL
LIN {X 0,Y 587.369,Z 154.798,A -85,B 0,C 180,E1 -1414.864,E2 -1414.864} C_VEL
LIN {X 0,Y 587.313,Z 163.113,A -85,B 0,C 180,E1 -1417.485,E2 -1417.485} C_VEL
LIN {X 0,Y 587.302,Z 171.417,A -85,B 0,C 180,E1 -1420.059,E2 -1420.059} C_VEL
LIN {X 0,Y 587.241,Z 179.698,A -85,B 0,C 180,E1 -1422.591,E2 -1422.591} C_VEL
LIN {X 0,Y 587.263,Z 189.163,A -85,B 0,C 180,E1 -1425.445,E2 -1425.445} C_VEL
LIN {X 0,Y 587.198,Z 198.628,A -85,B 0,C 180,E1 -1428.26,E2 -1428.26} C_VEL
LIN {X 0,Y 587.177,Z 208.093,A -85,B 0,C 180,E1 -1431.049,E2 -1431.049} C_VEL
LIN {X 0,Y 587.17,Z 214.379,A -85,B 0,C 180,E1 -1432.888,E2 -1432.888} C_VEL
LIN {X 0,Y 587.344,Z 223.499,A -85,B 0,C 180,E1 -1433.191,E2 -1433.191} C_VEL
LIN {X 0,Y 587.259,Z 232.995,A -85,B 0,C 180,E1 -1433.643,E2 -1433.643} C_VEL
LIN {X 0,Y 587.211,Z 241.022,A -85,B 0,C 180,E1 -1434.161,E2 -1434.161} C_VEL
LIN {X 0,Y 587.261,Z 249.043,A -85,B 0,C 180,E1 -1434.85,E2 -1434.85} C_VEL
LIN {X 0,Y 587.216,Z 255.218,A -85,B 0,C 180,E1 -1435.538,E2 -1435.538} C_VEL
LIN {X 0,Y 587.228,Z 260.078,A -85,B 0,C 180,E1 -1436.226,E2 -1436.226} C_VEL
LIN {X 0,Y 587.184,Z 263.826,A -85,B 0,C 180,E1 -1436.913,E2 -1436.913} C_VEL
LIN {X 0,Y 587.145,Z 267.832,A -85,B 0,C 180,E1 -1437.942,E2 -1437.942} C_VEL
LIN {X 0,Y 587.148,Z 269.574,A -85,B 0,C 180,E1 -1438.628,E2 -1438.628} C_VEL
LIN {X 0,Y 587.14,Z 270.618,A -85,B 0,C 180,E1 -1439.314,E2 -1439.314} C_VEL
LIN {X 0,Y 587.137,Z 270.996,A -85,B 0,C 180,E1 -1440,E2 -1440} C_VEL
LIN {X 0,Y 587.14,Z 270.712,A -85,B 0,C 180,E1 -1440.686,E2 -1440.686} C_VEL
LIN {X 0,Y 587.148,Z 269.764,A -85,B 0,C 180,E1 -1441.372,E2 -1441.372} C_VEL
LIN {X 0,Y 587.144,Z 268.124,A -85,B 0,C 180,E1 -1442.058,E2 -1442.058} C_VEL
LIN {X 0,Y 587.145,Z 265.739,A -85,B 0,C 180,E1 -1442.744,E2 -1442.744} C_VEL
LIN {X 0,Y 587.228,Z 260.609,A -85,B 0,C 180,E1 -1443.774,E2 -1443.774} C_VEL
LIN {X 0,Y 587.241,Z 254.542,A -85,B 0,C 180,E1 -1444.634,E2 -1444.634} C_VEL
LIN {X 0,Y 587.207,Z 248.23,A -85,B 0,C 180,E1 -1445.322,E2 -1445.322} C_VEL
LIN {X 0,Y 587.209,Z 241.076,A -85,B 0,C 180,E1 -1445.925,E2 -1445.925} C_VEL
LIN {X 0,Y 587.25,Z 232.815,A -85,B 0,C 180,E1 -1446.457,E2 -1446.457} C_VEL
LIN {X 0,Y 587.366,Z 223.048,A -85,B 0,C 180,E1 -1446.915,E2 -1446.915} C_VEL
LIN {X 0,Y 587.173,Z 214.391,A -85,B 0,C 180,E1 -1447.198,E2 -1447.198} C_VEL
LIN {X 0,Y 587.176,Z 206.032,A -85,B 0,C 180,E1 -1449.647,E2 -1449.647} C_VEL
LIN {X 0,Y 587.212,Z 196.564,A -85,B 0,C 180,E1 -1452.441,E2 -1452.441} C_VEL
LIN {X 0,Y 587.24,Z 187.096,A -85,B 0,C 180,E1 -1455.266,E2 -1455.266} C_VEL
LIN {X 0,Y 587.273,Z 178.81,A -85,B 0,C 180,E1 -1457.768,E2 -1457.768} C_VEL
LIN {X 0,Y 587.324,Z 169.358,A -85,B 0,C 180,E1 -1460.666,E2 -1460.666} C_VEL
LIN {X 0,Y 587.326,Z 159.799,A -85,B 0,C 180,E1 -1463.632,E2 -1463.632} C_VEL
LIN {X 0,Y 587.383,Z 150.151,A -85,B 0,C 180,E1 -1466.659,E2 -1466.659} C_VEL
LIN {X 0,Y 587.438,Z 141.38,A -85,B 0,C 180,E1 -1469.375,E2 -1469.375} C_VEL
LIN {X 0,Y 587.36,Z 139.324,A -85,B 0,C 180,E1 -1470.07,E2 -1470.07} C_VEL
LIN {X 0,Y 587.342,Z 139.328,A -85,B 0,C 180,E1 -1472.579,E2 -1472.579} C_VEL
LIN {X 0,Y 587.331,Z 139.328,A -85,B 0,C 180,E1 -1475.056,E2 -1475.056} C_VEL
LIN {X 0,Y 587.347,Z 139.325,A -85,B 0,C 180,E1 -1477.839,E2 -1477.839} C_VEL
LIN {X 0,Y 587.316,Z 139.331,A -85,B 0,C 180,E1 -1480.254,E2 -1480.254} C_VEL
LIN {X 0,Y 587.318,Z 139.328,A -85,B 0,C 180,E1 -1483.118,E2 -1483.118} C_VEL
LIN {X 0,Y 587.329,Z 139.327,A -85,B 0,C 180,E1 -1486.049,E2 -1486.049} C_VEL
LIN {X 0,Y 587.34,Z 139.327,A -85,B 0,C 180,E1 -1488.925,E2 -1488.925} C_VEL
LIN {X 0,Y 587.325,Z 139.328,A -85,B 0,C 180,E1 -1491.519,E2 -1491.519} C_VEL
LIN {X 0,Y 587.298,Z 139.331,A -85,B 0,C 180,E1 -1494.1,E2 -1494.1} C_VEL
LIN {X 0,Y 587.334,Z 139.329,A -85,B 0,C 180,E1 -1496.602,E2 -1496.602} C_VEL
LIN {X 0,Y 587.342,Z 139.326,A -85,B 0,C 180,E1 -1499.49,E2 -1499.49} C_VEL
LIN {X 0,Y 587.357,Z 139.326,A -85,B 0,C 180,E1 -1502.307,E2 -1502.307} C_VEL
LIN {X 0,Y 587.386,Z 139.455,A -85,B 0,C 180,E1 -1503.004,E2 -1503.004} C_VEL
LIN {X 0,Y 587.837,Z 143.011,A -85,B 0,C 180,E1 -1503.745,E2 -1503.745} C_VEL
LIN {X 0,Y 587.745,Z 154.977,A -85,B 0,C 180,E1 -1506.01,E2 -1506.01} C_VEL
LIN {X 0,Y 587.603,Z 171.152,A -85,B 0,C 180,E1 -1508.972,E2 -1508.972} C_VEL
LIN {X 0,Y 587.466,Z 186.352,A -85,B 0,C 180,E1 -1511.697,E2 -1511.697} C_VEL
LIN {X 0,Y 587.415,Z 201.552,A -85,B 0,C 180,E1 -1514.383,E2 -1514.383} C_VEL
LIN {X 0,Y 587.338,Z 217.765,A -85,B 0,C 180,E1 -1517.21,E2 -1517.21} C_VEL
LIN {X 0,Y 587.32,Z 221.013,A -85,B 0,C 180,E1 -1517.758,E2 -1517.758} C_VEL
LIN {X 0,Y 587.761,Z 225.547,A -85,B 0,C 180,E1 -1517.833,E2 -1517.833} C_VEL
LIN {X 0,Y 587.701,Z 238.662,A -85,B 0,C 180,E1 -1518.116,E2 -1518.116} C_VEL
LIN {X 0,Y 587.611,Z 251.633,A -85,B 0,C 180,E1 -1518.546,E2 -1518.546} C_VEL
LIN {X 0,Y 587.543,Z 262.909,A -85,B 0,C 180,E1 -1519.053,E2 -1519.053} C_VEL
LIN {X 0,Y 587.464,Z 273.568,A -85,B 0,C 180,E1 -1519.661,E2 -1519.661} C_VEL
LIN {X 0,Y 587.398,Z 284.462,A -85,B 0,C 180,E1 -1520.443,E2 -1520.443} C_VEL
LIN {X 0,Y 587.31,Z 295.102,A -85,B 0,C 180,E1 -1521.396,E2 -1521.396} C_VEL
LIN {X 0,Y 587.274,Z 302.952,A -85,B 0,C 180,E1 -1522.262,E2 -1522.262} C_VEL
LIN {X 0,Y 587.231,Z 309.462,A -85,B 0,C 180,E1 -1523.125,E2 -1523.125} C_VEL
LIN {X 0,Y 587.237,Z 315.861,A -85,B 0,C 180,E1 -1524.16,E2 -1524.16} C_VEL
LIN {X 0,Y 587.147,Z 320.946,A -85,B 0,C 180,E1 -1525.193,E2 -1525.193} C_VEL
LIN {X 0,Y 587.213,Z 324.892,A -85,B 0,C 180,E1 -1526.225,E2 -1526.225} C_VEL
LIN {X 0,Y 587.132,Z 327.806,A -85,B 0,C 180,E1 -1527.255,E2 -1527.255} C_VEL
LIN {X 0,Y 587.141,Z 329.198,A -85,B 0,C 180,E1 -1527.941,E2 -1527.941} C_VEL
LIN {X 0,Y 587.14,Z 330.784,A -85,B 0,C 180,E1 -1529.313,E2 -1529.313} C_VEL
LIN {X 0,Y 587.137,Z 331,A -85,B 0,C 180,E1 -1529.999,E2 -1529.999} C_VEL
LIN {X 0,Y 587.147,Z 330.187,A -85,B 0,C 180,E1 -1531.371,E2 -1531.371} C_VEL
LIN {X 0,Y 587.141,Z 329.203,A -85,B 0,C 180,E1 -1532.057,E2 -1532.057} C_VEL
LIN {X 0,Y 587.132,Z 327.812,A -85,B 0,C 180,E1 -1532.743,E2 -1532.743} C_VEL
LIN {X 0,Y 587.213,Z 324.9,A -85,B 0,C 180,E1 -1533.773,E2 -1533.773} C_VEL
LIN {X 0,Y 587.147,Z 320.954,A -85,B 0,C 180,E1 -1534.805,E2 -1534.805} C_VEL
LIN {X 0,Y 587.217,Z 314.884,A -85,B 0,C 180,E1 -1536.01,E2 -1536.01} C_VEL
LIN {X 0,Y 587.246,Z 308.246,A -85,B 0,C 180,E1 -1537.045,E2 -1537.045} C_VEL
LIN {X 0,Y 587.299,Z 300.001,A -85,B 0,C 180,E1 -1538.082,E2 -1538.082} C_VEL
LIN {X 0,Y 587.343,Z 291.551,A -85,B 0,C 180,E1 -1538.948,E2 -1538.948} C_VEL
LIN {X 0,Y 587.415,Z 281.112,A -85,B 0,C 180,E1 -1539.815,E2 -1539.815} C_VEL
LIN {X 0,Y 587.489,Z 270.777,A -85,B 0,C 180,E1 -1540.51,E2 -1540.51} C_VEL
LIN {X 0,Y 587.561,Z 259.057,A -85,B 0,C 180,E1 -1541.138,E2 -1541.138} C_VEL
LIN {X 0,Y 587.62,Z 246.661,A -85,B 0,C 180,E1 -1541.637,E2 -1541.637} C_VEL
LIN {X 0,Y 587.705,Z 233.487,A -85,B 0,C 180,E1 -1542.013,E2 -1542.013} C_VEL
LIN {X 0,Y 587.577,Z 222.688,A -85,B 0,C 180,E1 -1542.213,E2 -1542.213} C_VEL
LIN {X 0,Y 587.323,Z 220.818,A -85,B 0,C 180,E1 -1542.262,E2 -1542.262} C_VEL
LIN {X 0,Y 587.374,Z 204.605,A -85,B 0,C 180,E1 -1545.083,E2 -1545.083} C_VEL
LIN {X 0,Y 587.496,Z 189.405,A -85,B 0,C 180,E1 -1547.76,E2 -1547.76} C_VEL
LIN {X 0,Y 587.541,Z 174.205,A -85,B 0,C 180,E1 -1550.479,E2 -1550.479} C_VEL
LIN {X 0,Y 587.662,Z 160.616,A -85,B 0,C 180,E1 -1552.947,E2 -1552.947} C_VEL
LIN {X 0,Y 587.805,Z 145.883,A -85,B 0,C 180,E1 -1555.683,E2 -1555.683} C_VEL
LIN {X 0,Y 587.599,Z 140.848,A -85,B 0,C 180,E1 -1556.647,E2 -1556.647} C_VEL
LIN {X 0,Y 587.379,Z 139.321,A -85,B 0,C 180,E1 -1556.994,E2 -1556.994} C_VEL
LIN {X 0,Y 587.302,Z 139.329,A -85,B 0,C 180,E1 -1559.38,E2 -1559.38} C_VEL
LIN {X 0,Y 587.339,Z 139.322,A -85,B 0,C 180,E1 -1561.834,E2 -1561.834} C_VEL
LIN {X 0,Y 587.353,Z 139.323,A -85,B 0,C 180,E1 -1564.348,E2 -1564.348} C_VEL
LIN {X 0,Y 587.348,Z 139.32,A -85,B 0,C 180,E1 -1566.745,E2 -1566.745} C_VEL
LIN {X 0,Y 587.323,Z 139.327,A -85,B 0,C 180,E1 -1569.359,E2 -1569.359} C_VEL
LIN {X 0,Y 587.326,Z 139.324,A -85,B 0,C 180,E1 -1572.106,E2 -1572.106} C_VEL
LIN {X 0,Y 587.307,Z 139.325,A -85,B 0,C 180,E1 -1575.088,E2 -1575.088} C_VEL
LIN {X 0,Y 587.343,Z 139.322,A -85,B 0,C 180,E1 -1577.926,E2 -1577.926} C_VEL
LIN {X 0,Y 587.326,Z 139.327,A -85,B 0,C 180,E1 -1581.057,E2 -1581.057} C_VEL
LIN {X 0,Y 587.304,Z 139.325,A -85,B 0,C 180,E1 -1583.296,E2 -1583.296} C_VEL
LIN {X 0,Y 587.341,Z 139.326,A -85,B 0,C 180,E1 -1585.778,E2 -1585.778} C_VEL
LIN {X 0,Y 587.346,Z 139.32,A -85,B 0,C 180,E1 -1588.231,E2 -1588.231} C_VEL
LIN {X 0,Y 587.341,Z 139.327,A -85,B 0,C 180,E1 -1590.865,E2 -1590.865} C_VEL
LIN {X 0,Y 587.352,Z 139.32,A -85,B 0,C 180,E1 -1593.817,E2 -1593.817} C_VEL
LIN {X 0,Y 587.318,Z 139.331,A -85,B 0,C 180,E1 -1595.993,E2 -1595.993} C_VEL
LIN {X 0,Y 587.303,Z 139.326,A -85,B 0,C 180,E1 -1598.225,E2 -1598.225} C_VEL
LIN {X 0,Y 587.342,Z 139.326,A -85,B 0,C 180,E1 -1601.151,E2 -1601.151} C_VEL
LIN {X 0,Y 587.347,Z 139.32,A -85,B 0,C 180,E1 -1603.311,E2 -1603.311} C_VEL
LIN {X 0,Y 587.354,Z 139.325,A -85,B 0,C 180,E1 -1606.154,E2 -1606.154} C_VEL
LIN {X 0,Y 587.329,Z 139.323,A -85,B 0,C 180,E1 -1608.962,E2 -1608.962} C_VEL
LIN {X 0,Y 587.329,Z 139.322,A -85,B 0,C 180,E1 -1611.744,E2 -1611.744} C_VEL
LIN {X 0,Y 587.351,Z 139.326,A -85,B 0,C 180,E1 -1614.507,E2 -1614.507} C_VEL
LIN {X 0,Y 587.37,Z 139.318,A -85,B 0,C 180,E1 -1617.257,E2 -1617.257} C_VEL
LIN {X 0,Y 587.356,Z 139.32,A -85,B 0,C 180,E1 -1620,E2 -1620} C_VEL
LIN {X 0,Y 587.354,Z 139.325,A -85,B 0,C 180,E1 -1622.743,E2 -1622.743} C_VEL
LIN {X 0,Y 587.34,Z 139.321,A -85,B 0,C 180,E1 -1625.493,E2 -1625.493} C_VEL
LIN {X 0,Y 587.364,Z 139.32,A -85,B 0,C 180,E1 -1628.255,E2 -1628.255} C_VEL
LIN {X 0,Y 587.347,Z 139.326,A -85,B 0,C 180,E1 -1631.142,E2 -1631.142} C_VEL
LIN {X 0,Y 587.34,Z 139.323,A -85,B 0,C 180,E1 -1634.257,E2 -1634.257} C_VEL
LIN {X 0,Y 587.343,Z 139.321,A -85,B 0,C 180,E1 -1637.406,E2 -1637.406} C_VEL
LIN {X 0,Y 587.313,Z 139.326,A -85,B 0,C 180,E1 -1638.331,E2 -1638.331} C_VEL
LIN {X 0,Y 586.659,Z 139.406,A -85,B 0,C 180,E1 -1638.903,E2 -1638.903} C_VEL
LIN {X 0,Y 583.825,Z 139.766,A -85,B 0,C 180,E1 -1639.831,E2 -1639.831} C_VEL
LIN {X 0,Y 581.417,Z 140.07,A -85,B 0,C 180,E1 -1640.578,E2 -1640.578} C_VEL
LIN {X 0,Y 580.37,Z 140.198,A -85,B 0,C 180,E1 -1641.154,E2 -1641.154} C_VEL
LIN {X 0,Y 580.278,Z 140.206,A -85,B 0,C 180,E1 -1641.35,E2 -1641.35} C_VEL
LIN {X 0,Y 580.29,Z 140.2,A -85,B 0,C 180,E1 -1643.557,E2 -1643.557} C_VEL
LIN {X 0,Y 580.27,Z 140.209,A -85,B 0,C 180,E1 -1646.334,E2 -1646.334} C_VEL
LIN {X 0,Y 580.287,Z 140.201,A -85,B 0,C 180,E1 -1649.311,E2 -1649.311} C_VEL
LIN {X 0,Y 580.291,Z 140.199,A -85,B 0,C 180,E1 -1652.201,E2 -1652.201} C_VEL
LIN {X 0,Y 580.293,Z 140.205,A -85,B 0,C 180,E1 -1654.696,E2 -1654.696} C_VEL
LIN {X 0,Y 580.288,Z 140.199,A -85,B 0,C 180,E1 -1657.269,E2 -1657.269} C_VEL
LIN {X 0,Y 580.275,Z 140.202,A -85,B 0,C 180,E1 -1660.271,E2 -1660.271} C_VEL
LIN {X 0,Y 580.269,Z 140.203,A -85,B 0,C 180,E1 -1662.707,E2 -1662.707} C_VEL
LIN {X 0,Y 580.265,Z 140.202,A -85,B 0,C 180,E1 -1665.61,E2 -1665.61} C_VEL
LIN {X 0,Y 580.306,Z 140.203,A -85,B 0,C 180,E1 -1668.236,E2 -1668.236} C_VEL
LIN {X 0,Y 580.26,Z 140.203,A -85,B 0,C 180,E1 -1670.966,E2 -1670.966} C_VEL
LIN {X 0,Y 580.239,Z 140.207,A -85,B 0,C 180,E1 -1673.596,E2 -1673.596} C_VEL
LIN {X 0,Y 580.31,Z 140.198,A -85,B 0,C 180,E1 -1676.147,E2 -1676.147} C_VEL
LIN {X 0,Y 580.285,Z 140.202,A -85,B 0,C 180,E1 -1678.617,E2 -1678.617} C_VEL
LIN {X 0,Y 580.291,Z 140.2,A -85,B 0,C 180,E1 -1681.025,E2 -1681.025} C_VEL
LIN {X 0,Y 580.281,Z 140.202,A -85,B 0,C 180,E1 -1683.668,E2 -1683.668} C_VEL
LIN {X 0,Y 580.246,Z 140.209,A -85,B 0,C 180,E1 -1686.442,E2 -1686.442} C_VEL
LIN {X 0,Y 580.268,Z 140.203,A -85,B 0,C 180,E1 -1689.438,E2 -1689.438} C_VEL
LIN {X 0,Y 580.266,Z 140.209,A -85,B 0,C 180,E1 -1691.646,E2 -1691.646} C_VEL
LIN {X 0,Y 580.276,Z 140.202,A -85,B 0,C 180,E1 -1693.827,E2 -1693.827} C_VEL
LIN {X 0,Y 580.303,Z 140.197,A -85,B 0,C 180,E1 -1695.984,E2 -1695.984} C_VEL
LIN {X 0,Y 580.305,Z 140.198,A -85,B 0,C 180,E1 -1698.828,E2 -1698.828} C_VEL
LIN {X 0,Y 580.326,Z 140.201,A -85,B 0,C 180,E1 -1701.645,E2 -1701.645} C_VEL
LIN {X 0,Y 580.325,Z 140.195,A -85,B 0,C 180,E1 -1704.441,E2 -1704.441} C_VEL
LIN {X 0,Y 580.329,Z 140.196,A -85,B 0,C 180,E1 -1707.225,E2 -1707.225} C_VEL
LIN {X 0,Y 580.35,Z 140.197,A -85,B 0,C 180,E1 -1710.001,E2 -1710.001} C_VEL
LIN {X 0,Y 580.32,Z 140.195,A -85,B 0,C 180,E1 -1712.778,E2 -1712.778} C_VEL
LIN {X 0,Y 580.328,Z 140.196,A -85,B 0,C 180,E1 -1715.561,E2 -1715.561} C_VEL
LIN {X 0,Y 580.331,Z 140.199,A -85,B 0,C 180,E1 -1718.357,E2 -1718.357} C_VEL
LIN {X 0,Y 580.305,Z 140.197,A -85,B 0,C 180,E1 -1721.192,E2 -1721.192} C_VEL
LIN {X 0,Y 580.281,Z 140.201,A -85,B 0,C 180,E1 -1724.019,E2 -1724.019} C_VEL
LIN {X 0,Y 580.318,Z 140.202,A -85,B 0,C 180,E1 -1726.915,E2 -1726.915} C_VEL
LIN {X 0,Y 580.292,Z 140.201,A -85,B 0,C 180,E1 -1729.824,E2 -1729.824} C_VEL
LIN {X 0,Y 580.26,Z 140.208,A -85,B 0,C 180,E1 -1732.054,E2 -1732.054} C_VEL
LIN {X 0,Y 580.277,Z 140.205,A -85,B 0,C 180,E1 -1735.082,E2 -1735.082} C_VEL
LIN {X 0,Y 580.246,Z 140.206,A -85,B 0,C 180,E1 -1738.189,E2 -1738.189} C_VEL
LIN {X 0,Y 580.281,Z 140.203,A -85,B 0,C 180,E1 -1740.694,E2 -1740.694} C_VEL
LIN {X 0,Y 580.288,Z 140.202,A -85,B 0,C 180,E1 -1743.314,E2 -1743.314} C_VEL
LIN {X 0,Y 580.248,Z 140.206,A -85,B 0,C 180,E1 -1745.756,E2 -1745.756} C_VEL
LIN {X 0,Y 580.245,Z 140.205,A -85,B 0,C 180,E1 -1748.15,E2 -1748.15} C_VEL
LIN {X 0,Y 580.281,Z 140.202,A -85,B 0,C 180,E1 -1750.846,E2 -1750.846} C_VEL
LIN {X 0,Y 580.277,Z 140.207,A -85,B 0,C 180,E1 -1753.659,E2 -1753.659} C_VEL
LIN {X 0,Y 580.278,Z 140.202,A -85,B 0,C 180,E1 -1756.61,E2 -1756.61} C_VEL
LIN {X 0,Y 580.298,Z 140.2,A -85,B 0,C 180,E1 -1759.156,E2 -1759.156} C_VEL
LIN {X 0,Y 580.276,Z 140.204,A -85,B 0,C 180,E1 -1761.93,E2 -1761.93} C_VEL
LIN {X 0,Y 580.252,Z 140.204,A -85,B 0,C 180,E1 -1764.453,E2 -1764.453} C_VEL
LIN {X 0,Y 580.292,Z 140.203,A -85,B 0,C 180,E1 -1766.975,E2 -1766.975} C_VEL
LIN {X 0,Y 580.349,Z 140.332,A -85,B 0,C 180,E1 -1769.83,E2 -1769.83} C_VEL
LIN {X 0,Y 580.405,Z 147.307,A -85,B 0,C 180,E1 -1772.122,E2 -1772.122} C_VEL
LIN {X 0,Y 580.336,Z 155.963,A -85,B 0,C 180,E1 -1774.922,E2 -1774.922} C_VEL
LIN {X 0,Y 580.277,Z 164.3,A -85,B 0,C 180,E1 -1777.573,E2 -1777.573} C_VEL
LIN {X 0,Y 580.237,Z 172.639,A -85,B 0,C 180,E1 -1780.175,E2 -1780.175} C_VEL
LIN {X 0,Y 580.233,Z 182.11,A -85,B 0,C 180,E1 -1783.114,E2 -1783.114} C_VEL
LIN {X 0,Y 580.165,Z 191.531,A -85,B 0,C 180,E1 -1785.979,E2 -1785.979} C_VEL
LIN {X 0,Y 580.113,Z 200.996,A -85,B 0,C 180,E1 -1788.823,E2 -1788.823} C_VEL
LIN {X 0,Y 580.112,Z 210.461,A -85,B 0,C 180,E1 -1791.641,E2 -1791.641} C_VEL
LIN {X 0,Y 580.048,Z 214.381,A -85,B 0,C 180,E1 -1792.8,E2 -1792.8} C_VEL
LIN {X 0,Y 580.314,Z 221.76,A -85,B 0,C 180,E1 -1793.044,E2 -1793.044} C_VEL
LIN {X 0,Y 580.222,Z 230.755,A -85,B 0,C 180,E1 -1793.438,E2 -1793.438} C_VEL
LIN {X 0,Y 580.186,Z 238.587,A -85,B 0,C 180,E1 -1793.916,E2 -1793.916} C_VEL
LIN {X 0,Y 580.107,Z 245.311,A -85,B 0,C 180,E1 -1794.438,E2 -1794.438} C_VEL
LIN {X 0,Y 580.173,Z 252.373,A -85,B 0,C 180,E1 -1795.136,E2 -1795.136} C_VEL
LIN {X 0,Y 580.109,Z 257.763,A -85,B 0,C 180,E1 -1795.832,E2 -1795.832} C_VEL
LIN {X 0,Y 580.129,Z 262.026,A -85,B 0,C 180,E1 -1796.527,E2 -1796.527} C_VEL
LIN {X 0,Y 580.057,Z 265.344,A -85,B 0,C 180,E1 -1797.222,E2 -1797.222} C_VEL
LIN {X 0,Y 580.047,Z 267.835,A -85,B 0,C 180,E1 -1797.917,E2 -1797.917} C_VEL
LIN {X 0,Y 580.047,Z 269.576,A -85,B 0,C 180,E1 -1798.611,E2 -1798.611} C_VEL
LIN {X 0,Y 580.041,Z 270.62,A -85,B 0,C 180,E1 -1799.306,E2 -1799.306} C_VEL
LIN {X 0,Y 580.038,Z 270.996,A -85,B 0,C 180,E1 -1800,E2 -1800} C_VEL
LIN {X 0,Y 580.04,Z 270.712,A -85,B 0,C 180,E1 -1800.694,E2 -1800.694} C_VEL
LIN {X 0,Y 580.048,Z 269.763,A -85,B 0,C 180,E1 -1801.389,E2 -1801.389} C_VEL
LIN {X 0,Y 580.046,Z 268.122,A -85,B 0,C 180,E1 -1802.083,E2 -1802.083} C_VEL
LIN {X 0,Y 580.057,Z 265.737,A -85,B 0,C 180,E1 -1802.778,E2 -1802.778} C_VEL
LIN {X 0,Y 580.158,Z 260.607,A -85,B 0,C 180,E1 -1803.82,E2 -1803.82} C_VEL
LIN {X 0,Y 580.169,Z 254.537,A -85,B 0,C 180,E1 -1804.69,E2 -1804.69} C_VEL
LIN {X 0,Y 580.116,Z 248.223,A -85,B 0,C 180,E1 -1805.387,E2 -1805.387} C_VEL
LIN {X 0,Y 580.16,Z 241.07,A -85,B 0,C 180,E1 -1805.997,E2 -1805.997} C_VEL
LIN {X 0,Y 580.211,Z 232.845,A -85,B 0,C 180,E1 -1806.534,E2 -1806.534} C_VEL
LIN {X 0,Y 580.329,Z 223.035,A -85,B 0,C 180,E1 -1807,E2 -1807} C_VEL
LIN {X 0,Y 580.129,Z 215.344,A -85,B 0,C 180,E1 -1807.253,E2 -1807.253} C_VEL
LIN {X 0,Y 580.071,Z 214.315,A -85,B 0,C 180,E1 -1807.309,E2 -1807.309} C_VEL
LIN {X 0,Y 580.109,Z 204.847,A -85,B 0,C 180,E1 -1810.118,E2 -1810.118} C_VEL
LIN {X 0,Y 580.143,Z 195.379,A -85,B 0,C 180,E1 -1812.951,E2 -1812.951} C_VEL
LIN {X 0,Y 580.176,Z 187.094,A -85,B 0,C 180,E1 -1815.456,E2 -1815.456} C_VEL
LIN {X 0,Y 580.206,Z 178.808,A -85,B 0,C 180,E1 -1817.992,E2 -1817.992} C_VEL
LIN {X 0,Y 580.271,Z 170.615,A -85,B 0,C 180,E1 -1820.563,E2 -1820.563} C_VEL
LIN {X 0,Y 580.284,Z 160.984,A -85,B 0,C 180,E1 -1823.558,E2 -1823.558} C_VEL
LIN {X 0,Y 580.36,Z 152.136,A -85,B 0,C 180,E1 -1826.347,E2 -1826.347} C_VEL
LIN {X 0,Y 580.438,Z 142.658,A -85,B 0,C 180,E1 -1829.333,E2 -1829.333} C_VEL
LIN {X 0,Y 580.343,Z 140.199,A -85,B 0,C 180,E1 -1830.17,E2 -1830.17} C_VEL
LIN {X 0,Y 580.293,Z 140.204,A -85,B 0,C 180,E1 -1833.025,E2 -1833.025} C_VEL
LIN {X 0,Y 580.252,Z 140.21,A -85,B 0,C 180,E1 -1835.756,E2 -1835.756} C_VEL
LIN {X 0,Y 580.293,Z 140.206,A -85,B 0,C 180,E1 -1838.146,E2 -1838.146} C_VEL
LIN {X 0,Y 580.302,Z 140.202,A -85,B 0,C 180,E1 -1840.843,E2 -1840.843} C_VEL
LIN {X 0,Y 580.277,Z 140.207,A -85,B 0,C 180,E1 -1843.658,E2 -1843.658} C_VEL
LIN {X 0,Y 580.283,Z 140.205,A -85,B 0,C 180,E1 -1846.609,E2 -1846.609} C_VEL
LIN {X 0,Y 580.302,Z 140.204,A -85,B 0,C 180,E1 -1849.156,E2 -1849.156} C_VEL
LIN {X 0,Y 580.292,Z 140.204,A -85,B 0,C 180,E1 -1851.927,E2 -1851.927} C_VEL
LIN {X 0,Y 580.262,Z 140.21,A -85,B 0,C 180,E1 -1854.453,E2 -1854.453} C_VEL
LIN {X 0,Y 580.295,Z 140.204,A -85,B 0,C 180,E1 -1856.975,E2 -1856.975} C_VEL
LIN {X 0,Y 580.302,Z 140.204,A -85,B 0,C 180,E1 -1859.425,E2 -1859.425} C_VEL
LIN {X 0,Y 580.302,Z 140.206,A -85,B 0,C 180,E1 -1862.141,E2 -1862.141} C_VEL
LIN {X 0,Y 580.341,Z 140.261,A -85,B 0,C 180,E1 -1862.747,E2 -1862.747} C_VEL
LIN {X 0,Y 580.961,Z 145.484,A -85,B 0,C 180,E1 -1863.864,E2 -1863.864} C_VEL
LIN {X 0,Y 580.77,Z 159.101,A -85,B 0,C 180,E1 -1866.462,E2 -1866.462} C_VEL
LIN {X 0,Y 580.598,Z 173.285,A -85,B 0,C 180,E1 -1869.097,E2 -1869.097} C_VEL
LIN {X 0,Y 580.473,Z 187.365,A -85,B 0,C 180,E1 -1871.651,E2 -1871.651} C_VEL
LIN {X 0,Y 580.402,Z 202.565,A -85,B 0,C 180,E1 -1874.369,E2 -1874.369} C_VEL
LIN {X 0,Y 580.281,Z 218.779,A -85,B 0,C 180,E1 -1877.229,E2 -1877.229} C_VEL
LIN {X 0,Y 580.286,Z 221.013,A -85,B 0,C 180,E1 -1877.607,E2 -1877.607} C_VEL
LIN {X 0,Y 580.832,Z 226.896,A -85,B 0,C 180,E1 -1877.708,E2 -1877.708} C_VEL
LIN {X 0,Y 580.753,Z 239.424,A -85,B 0,C 180,E1 -1877.994,E2 -1877.994} C_VEL
LIN {X 0,Y 580.652,Z 252.349,A -85,B 0,C 180,E1 -1878.435,E2 -1878.435} C_VEL
LIN {X 0,Y 580.584,Z 264.611,A -85,B 0,C 180,E1 -1879.008,E2 -1879.008} C_VEL
LIN {X 0,Y 580.422,Z 276.188,A -85,B 0,C 180,E1 -1879.711,E2 -1879.711} C_VEL
LIN {X 0,Y 580.347,Z 286.588,A -85,B 0,C 180,E1 -1880.502,E2 -1880.502} C_VEL
LIN {X 0,Y 580.267,Z 295.102,A -85,B 0,C 180,E1 -1881.291,E2 -1881.291} C_VEL
LIN {X 0,Y 580.222,Z 302.952,A -85,B 0,C 180,E1 -1882.167,E2 -1882.167} C_VEL
LIN {X 0,Y 580.155,Z 310.646,A -85,B 0,C 180,E1 -1883.221,E2 -1883.221} C_VEL
LIN {X 0,Y 580.139,Z 317.675,A -85,B 0,C 180,E1 -1884.437,E2 -1884.437} C_VEL
LIN {X 0,Y 580.108,Z 322.368,A -85,B 0,C 180,E1 -1885.482,E2 -1885.482} C_VEL
LIN {X 0,Y 580.123,Z 325.954,A -85,B 0,C 180,E1 -1886.526,E2 -1886.526} C_VEL
LIN {X 0,Y 580.043,Z 327.806,A -85,B 0,C 180,E1 -1887.221,E2 -1887.221} C_VEL
LIN {X 0,Y 580.04,Z 329.197,A -85,B 0,C 180,E1 -1887.916,E2 -1887.916} C_VEL
LIN {X 0,Y 580.04,Z 330.784,A -85,B 0,C 180,E1 -1889.305,E2 -1889.305} C_VEL
LIN {X 0,Y 580.037,Z 331,A -85,B 0,C 180,E1 -1889.999,E2 -1889.999} C_VEL
LIN {X 0,Y 580.047,Z 330.187,A -85,B 0,C 180,E1 -1891.387,E2 -1891.387} C_VEL
LIN {X 0,Y 580.04,Z 329.202,A -85,B 0,C 180,E1 -1892.082,E2 -1892.082} C_VEL
LIN {X 0,Y 580.043,Z 327.812,A -85,B 0,C 180,E1 -1892.777,E2 -1892.777} C_VEL
LIN {X 0,Y 580.109,Z 324.9,A -85,B 0,C 180,E1 -1893.819,E2 -1893.819} C_VEL
LIN {X 0,Y 580.053,Z 320.954,A -85,B 0,C 180,E1 -1894.864,E2 -1894.864} C_VEL
LIN {X 0,Y 580.165,Z 315.873,A -85,B 0,C 180,E1 -1895.909,E2 -1895.909} C_VEL
LIN {X 0,Y 580.184,Z 308.246,A -85,B 0,C 180,E1 -1897.131,E2 -1897.131} C_VEL
LIN {X 0,Y 580.25,Z 300.001,A -85,B 0,C 180,E1 -1898.181,E2 -1898.181} C_VEL
LIN {X 0,Y 580.307,Z 291.551,A -85,B 0,C 180,E1 -1899.057,E2 -1899.057} C_VEL
LIN {X 0,Y 580.415,Z 281.113,A -85,B 0,C 180,E1 -1899.935,E2 -1899.935} C_VEL
LIN {X 0,Y 580.506,Z 269.348,A -85,B 0,C 180,E1 -1900.726,E2 -1900.726} C_VEL
LIN {X 0,Y 580.622,Z 256.828,A -85,B 0,C 180,E1 -1901.373,E2 -1901.373} C_VEL
LIN {X 0,Y 580.685,Z 245.21,A -85,B 0,C 180,E1 -1901.828,E2 -1901.828} C_VEL
LIN {X 0,Y 580.773,Z 232.572,A -85,B 0,C 180,E1 -1902.18,E2 -1902.18} C_VEL
LIN {X 0,Y 580.647,Z 223.442,A -85,B 0,C 180,E1 -1902.349,E2 -1902.349} C_VEL
LIN {X 0,Y 580.27,Z 220.818,A -85,B 0,C 180,E1 -1902.413,E2 -1902.413} C_VEL
LIN {X 0,Y 580.347,Z 205.618,A -85,B 0,C 180,E1 -1905.09,E2 -1905.09} C_VEL
LIN {X 0,Y 580.504,Z 190.418,A -85,B 0,C 180,E1 -1907.799,E2 -1907.799} C_VEL
LIN {X 0,Y 580.569,Z 175.218,A -85,B 0,C 180,E1 -1910.55,E2 -1910.55} C_VEL
LIN {X 0,Y 580.715,Z 161.343,A -85,B 0,C 180,E1 -1913.106,E2 -1913.106} C_VEL
LIN {X 0,Y 580.89,Z 146.942,A -85,B 0,C 180,E1 -1915.819,E2 -1915.819} C_VEL
LIN {X 0,Y 580.619,Z 141.906,A -85,B 0,C 180,E1 -1916.799,E2 -1916.799} C_VEL
LIN {X 0,Y 580.329,Z 140.201,A -85,B 0,C 180,E1 -1917.154,E2 -1917.154} C_VEL
LIN {X 0,Y 580.255,Z 140.205,A -85,B 0,C 180,E1 -1919.773,E2 -1919.773} C_VEL
LIN {X 0,Y 580.294,Z 140.203,A -85,B 0,C 180,E1 -1922.199,E2 -1922.199} C_VEL
LIN {X 0,Y 580.298,Z 140.199,A -85,B 0,C 180,E1 -1924.694,E2 -1924.694} C_VEL
LIN {X 0,Y 580.294,Z 140.203,A -85,B 0,C 180,E1 -1927.267,E2 -1927.267} C_VEL
LIN {X 0,Y 580.278,Z 140.201,A -85,B 0,C 180,E1 -1930.269,E2 -1930.269} C_VEL
LIN {X 0,Y 580.261,Z 140.206,A -85,B 0,C 180,E1 -1932.706,E2 -1932.706} C_VEL
LIN {X 0,Y 580.265,Z 140.206,A -85,B 0,C 180,E1 -1935.607,E2 -1935.607} C_VEL
LIN {X 0,Y 580.305,Z 140.197,A -85,B 0,C 180,E1 -1938.233,E2 -1938.233} C_VEL
LIN {X 0,Y 580.282,Z 140.206,A -85,B 0,C 180,E1 -1940.965,E2 -1940.965} C_VEL
LIN {X 0,Y 580.233,Z 140.206,A -85,B 0,C 180,E1 -1943.594,E2 -1943.594} C_VEL
LIN {X 0,Y 580.3,Z 140.202,A -85,B 0,C 180,E1 -1946.144,E2 -1946.144} C_VEL
LIN {X 0,Y 580.281,Z 140.2,A -85,B 0,C 180,E1 -1948.615,E2 -1948.615} C_VEL
LIN {X 0,Y 580.285,Z 140.206,A -85,B 0,C 180,E1 -1951.023,E2 -1951.023} C_VEL
LIN {X 0,Y 580.317,Z 140.196,A -85,B 0,C 180,E1 -1953.657,E2 -1953.657} C_VEL
LIN {X 0,Y 580.259,Z 140.204,A -85,B 0,C 180,E1 -1956.441,E2 -1956.441} C_VEL
LIN {X 0,Y 580.265,Z 140.208,A -85,B 0,C 180,E1 -1959.437,E2 -1959.437} C_VEL
LIN {X 0,Y 580.274,Z 140.202,A -85,B 0,C 180,E1 -1961.645,E2 -1961.645} C_VEL
LIN {X 0,Y 580.274,Z 140.202,A -85,B 0,C 180,E1 -1963.825,E2 -1963.825} C_VEL
LIN {X 0,Y 580.323,Z 140.201,A -85,B 0,C 180,E1 -1965.983,E2 -1965.983} C_VEL
LIN {X 0,Y 580.289,Z 140.199,A -85,B 0,C 180,E1 -1968.826,E2 -1968.826} C_VEL
LIN {X 0,Y 580.299,Z 140.199,A -85,B 0,C 180,E1 -1971.643,E2 -1971.643} C_VEL
LIN {X 0,Y 580.315,Z 140.202,A -85,B 0,C 180,E1 -1974.44,E2 -1974.44} C_VEL
LIN {X 0,Y 580.336,Z 140.194,A -85,B 0,C 180,E1 -1977.223,E2 -1977.223} C_VEL
LIN {X 0,Y 580.326,Z 140.195,A -85,B 0,C 180,E1 -1980,E2 -1980} C_VEL
LIN {X 0,Y 580.32,Z 140.201,A -85,B 0,C 180,E1 -1982.777,E2 -1982.777} C_VEL
LIN {X 0,Y 580.306,Z 140.197,A -85,B 0,C 180,E1 -1985.56,E2 -1985.56} C_VEL
LIN {X 0,Y 580.327,Z 140.196,A -85,B 0,C 180,E1 -1988.356,E2 -1988.356} C_VEL
LIN {X 0,Y 580.318,Z 140.202,A -85,B 0,C 180,E1 -1991.209,E2 -1991.209} C_VEL
LIN {X 0,Y 580.292,Z 140.202,A -85,B 0,C 180,E1 -1994.336,E2 -1994.336} C_VEL
LIN {X 0,Y 580.301,Z 140.198,A -85,B 0,C 180,E1 -1996.916,E2 -1996.916} C_VEL
LIN {X 0,Y 580.296,Z 140.203,A -85,B 0,C 180,E1 -1999.823,E2 -1999.823} C_VEL
LIN {X 0,Y 580.278,Z 140.206,A -85,B 0,C 180,E1 -2001.35,E2 -2001.35} C_VEL
LIN {X 0,Y 579.588,Z 140.289,A -85,B 0,C 180,E1 -2001.929,E2 -2001.929} C_VEL
LIN {X 0,Y 576.715,Z 140.65,A -85,B 0,C 180,E1 -2002.869,E2 -2002.869} C_VEL
LIN {X 0,Y 574.316,Z 140.945,A -85,B 0,C 180,E1 -2003.626,E2 -2003.626} C_VEL
LIN {X 0,Y 573.31,Z 141.07,A -85,B 0,C 180,E1 -2004.21,E2 -2004.21} C_VEL
LIN {X 0,Y 573.241,Z 141.081,A -85,B 0,C 180,E1 -2004.407,E2 -2004.407} C_VEL
LIN {X 0,Y 573.182,Z 141.084,A -85,B 0,C 180,E1 -2006.979,E2 -2006.979} C_VEL
LIN {X 0,Y 573.235,Z 141.082,A -85,B 0,C 180,E1 -2009.489,E2 -2009.489} C_VEL
LIN {X 0,Y 573.243,Z 141.077,A -85,B 0,C 180,E1 -2012.23,E2 -2012.23} C_VEL
LIN {X 0,Y 573.244,Z 141.083,A -85,B 0,C 180,E1 -2014.775,E2 -2014.775} C_VEL
LIN {X 0,Y 573.242,Z 141.077,A -85,B 0,C 180,E1 -2017.167,E2 -2017.167} C_VEL
LIN {X 0,Y 573.226,Z 141.084,A -85,B 0,C 180,E1 -2019.609,E2 -2019.609} C_VEL
LIN {X 0,Y 573.231,Z 141.079,A -85,B 0,C 180,E1 -2022.643,E2 -2022.643} C_VEL
LIN {X 0,Y 573.23,Z 141.079,A -85,B 0,C 180,E1 -2025.668,E2 -2025.668} C_VEL
LIN {X 0,Y 573.237,Z 141.08,A -85,B 0,C 180,E1 -2028.546,E2 -2028.546} C_VEL
LIN {X 0,Y 573.227,Z 141.083,A -85,B 0,C 180,E1 -2031.299,E2 -2031.299} C_VEL
LIN {X 0,Y 573.184,Z 141.084,A -85,B 0,C 180,E1 -2034.023,E2 -2034.023} C_VEL
LIN {X 0,Y 573.279,Z 141.079,A -85,B 0,C 180,E1 -2036.52,E2 -2036.52} C_VEL
LIN {X 0,Y 573.24,Z 141.077,A -85,B 0,C 180,E1 -2039.116,E2 -2039.116} C_VEL
LIN {X 0,Y 573.249,Z 141.078,A -85,B 0,C 180,E1 -2041.972,E2 -2041.972} C_VEL
LIN {X 0,Y 573.227,Z 141.081,A -85,B 0,C 180,E1 -2044.59,E2 -2044.59} C_VEL
LIN {X 0,Y 573.217,Z 141.08,A -85,B 0,C 180,E1 -2047.663,E2 -2047.663} C_VEL
LIN {X 0,Y 573.273,Z 141.073,A -85,B 0,C 180,E1 -2050.672,E2 -2050.672} C_VEL
LIN {X 0,Y 573.249,Z 141.079,A -85,B 0,C 180,E1 -2053.623,E2 -2053.623} C_VEL
LIN {X 0,Y 573.249,Z 141.076,A -85,B 0,C 180,E1 -2055.808,E2 -2055.808} C_VEL
LIN {X 0,Y 573.263,Z 141.076,A -85,B 0,C 180,E1 -2058.746,E2 -2058.746} C_VEL
LIN {X 0,Y 573.281,Z 141.077,A -85,B 0,C 180,E1 -2061.542,E2 -2061.542} C_VEL
LIN {X 0,Y 573.292,Z 141.071,A -85,B 0,C 180,E1 -2064.373,E2 -2064.373} C_VEL
LIN {X 0,Y 573.312,Z 141.069,A -85,B 0,C 180,E1 -2067.894,E2 -2067.894} C_VEL
LIN {X 0,Y 573.319,Z 141.073,A -85,B 0,C 180,E1 -2070.001,E2 -2070.001} C_VEL
LIN {X 0,Y 573.289,Z 141.071,A -85,B 0,C 180,E1 -2072.812,E2 -2072.812} C_VEL
LIN {X 0,Y 573.295,Z 141.072,A -85,B 0,C 180,E1 -2075.629,E2 -2075.629} C_VEL
LIN {X 0,Y 573.286,Z 141.078,A -85,B 0,C 180,E1 -2078.46,E2 -2078.46} C_VEL
LIN {X 0,Y 573.276,Z 141.073,A -85,B 0,C 180,E1 -2081.313,E2 -2081.313} C_VEL
LIN {X 0,Y 573.246,Z 141.076,A -85,B 0,C 180,E1 -2084.41,E2 -2084.41} C_VEL
LIN {X 0,Y 573.263,Z 141.079,A -85,B 0,C 180,E1 -2087.112,E2 -2087.112} C_VEL
LIN {X 0,Y 573.246,Z 141.081,A -85,B 0,C 180,E1 -2090.078,E2 -2090.078} C_VEL
LIN {X 0,Y 573.226,Z 141.081,A -85,B 0,C 180,E1 -2092.339,E2 -2092.339} C_VEL
LIN {X 0,Y 573.224,Z 141.084,A -85,B 0,C 180,E1 -2095.412,E2 -2095.412} C_VEL
LIN {X 0,Y 573.208,Z 141.087,A -85,B 0,C 180,E1 -2098.567,E2 -2098.567} C_VEL
LIN {X 0,Y 573.226,Z 141.079,A -85,B 0,C 180,E1 -2100.994,E2 -2100.994} C_VEL
LIN {X 0,Y 573.246,Z 141.082,A -85,B 0,C 180,E1 -2103.521,E2 -2103.521} C_VEL
LIN {X 0,Y 573.197,Z 141.083,A -85,B 0,C 180,E1 -2106.054,E2 -2106.054} C_VEL
LIN {X 0,Y 573.22,Z 141.087,A -85,B 0,C 180,E1 -2108.704,E2 -2108.704} C_VEL
LIN {X 0,Y 573.213,Z 141.081,A -85,B 0,C 180,E1 -2111.459,E2 -2111.459} C_VEL
LIN {X 0,Y 573.243,Z 141.083,A -85,B 0,C 180,E1 -2113.669,E2 -2113.669} C_VEL
LIN {X 0,Y 573.24,Z 141.079,A -85,B 0,C 180,E1 -2116.641,E2 -2116.641} C_VEL
LIN {X 0,Y 573.25,Z 141.076,A -85,B 0,C 180,E1 -2119.475,E2 -2119.475} C_VEL
LIN {X 0,Y 573.218,Z 141.087,A -85,B 0,C 180,E1 -2122.191,E2 -2122.191} C_VEL
LIN {X 0,Y 573.235,Z 141.081,A -85,B 0,C 180,E1 -2125.23,E2 -2125.23} C_VEL
LIN {X 0,Y 573.244,Z 141.078,A -85,B 0,C 180,E1 -2128.185,E2 -2128.185} C_VEL
LIN {X 0,Y 573.288,Z 141.195,A -85,B 0,C 180,E1 -2129.725,E2 -2129.725} C_VEL
LIN {X 0,Y 573.42,Z 146.331,A -85,B 0,C 180,E1 -2131.445,E2 -2131.445} C_VEL
LIN {X 0,Y 573.319,Z 154.751,A -85,B 0,C 180,E1 -2134.204,E2 -2134.204} C_VEL
LIN {X 0,Y 573.24,Z 163.094,A -85,B 0,C 180,E1 -2136.901,E2 -2136.901} C_VEL
LIN {X 0,Y 573.217,Z 171.546,A -85,B 0,C 180,E1 -2139.548,E2 -2139.548} C_VEL
LIN {X 0,Y 573.141,Z 179.743,A -85,B 0,C 180,E1 -2142.148,E2 -2142.148} C_VEL
LIN {X 0,Y 573.108,Z 187.983,A -85,B 0,C 180,E1 -2144.713,E2 -2144.713} C_VEL
LIN {X 0,Y 573.081,Z 196.265,A -85,B 0,C 180,E1 -2147.247,E2 -2147.247} C_VEL
LIN {X 0,Y 573.016,Z 205.73,A -85,B 0,C 180,E1 -2150.113,E2 -2150.113} C_VEL
LIN {X 0,Y 572.985,Z 214.383,A -85,B 0,C 180,E1 -2152.711,E2 -2152.711} C_VEL
LIN {X 0,Y 573.28,Z 221.775,A -85,B 0,C 180,E1 -2152.958,E2 -2152.958} C_VEL
LIN {X 0,Y 573.198,Z 230.198,A -85,B 0,C 180,E1 -2153.328,E2 -2153.328} C_VEL
LIN {X 0,Y 573.127,Z 238.592,A -85,B 0,C 180,E1 -2153.84,E2 -2153.84} C_VEL
LIN {X 0,Y 573.047,Z 245.318,A -85,B 0,C 180,E1 -2154.369,E2 -2154.369} C_VEL
LIN {X 0,Y 573.09,Z 252.378,A -85,B 0,C 180,E1 -2155.076,E2 -2155.076} C_VEL
LIN {X 0,Y 573.037,Z 257.767,A -85,B 0,C 180,E1 -2155.78,E2 -2155.78} C_VEL
LIN {X 0,Y 573.062,Z 262.029,A -85,B 0,C 180,E1 -2156.484,E2 -2156.484} C_VEL
LIN {X 0,Y 572.973,Z 265.347,A -85,B 0,C 180,E1 -2157.188,E2 -2157.188} C_VEL
LIN {X 0,Y 572.951,Z 267.837,A -85,B 0,C 180,E1 -2157.891,E2 -2157.891} C_VEL
LIN {X 0,Y 572.947,Z 269.578,A -85,B 0,C 180,E1 -2158.594,E2 -2158.594} C_VEL
LIN {X 0,Y 572.941,Z 270.621,A -85,B 0,C 180,E1 -2159.297,E2 -2159.297} C_VEL
LIN {X 0,Y 572.938,Z 270.996,A -85,B 0,C 180,E1 -2160,E2 -2160} C_VEL
LIN {X 0,Y 572.941,Z 270.711,A -85,B 0,C 180,E1 -2160.703,E2 -2160.703} C_VEL
LIN {X 0,Y 572.948,Z 269.762,A -85,B 0,C 180,E1 -2161.406,E2 -2161.406} C_VEL
LIN {X 0,Y 572.95,Z 268.121,A -85,B 0,C 180,E1 -2162.109,E2 -2162.109} C_VEL
LIN {X 0,Y 572.973,Z 265.734,A -85,B 0,C 180,E1 -2162.812,E2 -2162.812} C_VEL
LIN {X 0,Y 573.085,Z 260.604,A -85,B 0,C 180,E1 -2163.868,E2 -2163.868} C_VEL
LIN {X 0,Y 573.097,Z 254.531,A -85,B 0,C 180,E1 -2164.748,E2 -2164.748} C_VEL
LIN {X 0,Y 573.032,Z 248.217,A -85,B 0,C 180,E1 -2165.454,E2 -2165.454} C_VEL
LIN {X 0,Y 573.117,Z 241.064,A -85,B 0,C 180,E1 -2166.071,E2 -2166.071} C_VEL
LIN {X 0,Y 573.156,Z 232.931,A -85,B 0,C 180,E1 -2166.609,E2 -2166.609} C_VEL
LIN {X 0,Y 573.259,Z 224.192,A -85,B 0,C 180,E1 -2167.042,E2 -2167.042} C_VEL
LIN {X 0,Y 573.08,Z 215.739,A -85,B 0,C 180,E1 -2167.332,E2 -2167.332} C_VEL
LIN {X 0,Y 572.983,Z 214.313,A -85,B 0,C 180,E1 -2167.4,E2 -2167.4} C_VEL
LIN {X 0,Y 573.013,Z 206.029,A -85,B 0,C 180,E1 -2169.887,E2 -2169.887} C_VEL
LIN {X 0,Y 573.081,Z 196.56,A -85,B 0,C 180,E1 -2172.753,E2 -2172.753} C_VEL
LIN {X 0,Y 573.105,Z 188.275,A -85,B 0,C 180,E1 -2175.287,E2 -2175.287} C_VEL
LIN {X 0,Y 573.184,Z 178.882,A -85,B 0,C 180,E1 -2178.22,E2 -2178.22} C_VEL
LIN {X 0,Y 573.233,Z 170.677,A -85,B 0,C 180,E1 -2180.827,E2 -2180.827} C_VEL
LIN {X 0,Y 573.275,Z 160.982,A -85,B 0,C 180,E1 -2183.864,E2 -2183.864} C_VEL
LIN {X 0,Y 573.345,Z 151.211,A -85,B 0,C 180,E1 -2186.971,E2 -2186.971} C_VEL
LIN {X 0,Y 573.436,Z 143.216,A -85,B 0,C 180,E1 -2189.52,E2 -2189.52} C_VEL
LIN {X 0,Y 573.296,Z 141.077,A -85,B 0,C 180,E1 -2190.275,E2 -2190.275} C_VEL
LIN {X 0,Y 573.258,Z 141.082,A -85,B 0,C 180,E1 -2192.645,E2 -2192.645} C_VEL
LIN {X 0,Y 573.213,Z 141.086,A -85,B 0,C 180,E1 -2195.188,E2 -2195.188} C_VEL
LIN {X 0,Y 573.241,Z 141.082,A -85,B 0,C 180,E1 -2197.807,E2 -2197.807} C_VEL
LIN {X 0,Y 573.25,Z 141.081,A -85,B 0,C 180,E1 -2200.525,E2 -2200.525} C_VEL
LIN {X 0,Y 573.241,Z 141.082,A -85,B 0,C 180,E1 -2203.359,E2 -2203.359} C_VEL
LIN {X 0,Y 573.25,Z 141.08,A -85,B 0,C 180,E1 -2206.331,E2 -2206.331} C_VEL
LIN {X 0,Y 573.239,Z 141.081,A -85,B 0,C 180,E1 -2208.543,E2 -2208.543} C_VEL
LIN {X 0,Y 573.243,Z 141.084,A -85,B 0,C 180,E1 -2211.298,E2 -2211.298} C_VEL
LIN {X 0,Y 573.22,Z 141.084,A -85,B 0,C 180,E1 -2214.018,E2 -2214.018} C_VEL
LIN {X 0,Y 573.245,Z 141.083,A -85,B 0,C 180,E1 -2216.515,E2 -2216.515} C_VEL
LIN {X 0,Y 573.235,Z 141.085,A -85,B 0,C 180,E1 -2219.117,E2 -2219.117} C_VEL
LIN {X 0,Y 573.254,Z 141.084,A -85,B 0,C 180,E1 -2221.971,E2 -2221.971} C_VEL
LIN {X 0,Y 573.303,Z 141.273,A -85,B 0,C 180,E1 -2222.532,E2 -2222.532} C_VEL
LIN {X 0,Y 574.063,Z 146.187,A -85,B 0,C 180,E1 -2223.604,E2 -2223.604} C_VEL
LIN {X 0,Y 573.874,Z 158.205,A -85,B 0,C 180,E1 -2225.97,E2 -2225.97} C_VEL
LIN {X 0,Y 573.627,Z 173.581,A -85,B 0,C 180,E1 -2228.892,E2 -2228.892} C_VEL
LIN {X 0,Y 573.471,Z 188.379,A -85,B 0,C 180,E1 -2231.604,E2 -2231.604} C_VEL
LIN {X 0,Y 573.367,Z 203.579,A -85,B 0,C 180,E1 -2234.355,E2 -2234.355} C_VEL
LIN {X 0,Y 573.227,Z 219.792,A -85,B 0,C 180,E1 -2237.25,E2 -2237.25} C_VEL
LIN {X 0,Y 573.232,Z 221.014,A -85,B 0,C 180,E1 -2237.452,E2 -2237.452} C_VEL
LIN {X 0,Y 573.892,Z 226.896,A -85,B 0,C 180,E1 -2237.557,E2 -2237.557} C_VEL
LIN {X 0,Y 573.817,Z 239.423,A -85,B 0,C 180,E1 -2237.847,E2 -2237.847} C_VEL
LIN {X 0,Y 573.678,Z 252.351,A -85,B 0,C 180,E1 -2238.293,E2 -2238.293} C_VEL
LIN {X 0,Y 573.577,Z 263.568,A -85,B 0,C 180,E1 -2238.816,E2 -2238.816} C_VEL
LIN {X 0,Y 573.466,Z 274.894,A -85,B 0,C 180,E1 -2239.495,E2 -2239.495} C_VEL
LIN {X 0,Y 573.352,Z 285.529,A -85,B 0,C 180,E1 -2240.296,E2 -2240.296} C_VEL
LIN {X 0,Y 573.239,Z 295.103,A -85,B 0,C 180,E1 -2241.184,E2 -2241.184} C_VEL
LIN {X 0,Y 573.162,Z 302.952,A -85,B 0,C 180,E1 -2242.07,E2 -2242.07} C_VEL
LIN {X 0,Y 573.074,Z 310.95,A -85,B 0,C 180,E1 -2243.185,E2 -2243.185} C_VEL
LIN {X 0,Y 573.071,Z 317.675,A -85,B 0,C 180,E1 -2244.369,E2 -2244.369} C_VEL
LIN {X 0,Y 573.029,Z 322.368,A -85,B 0,C 180,E1 -2245.426,E2 -2245.426} C_VEL
LIN {X 0,Y 573.022,Z 325.954,A -85,B 0,C 180,E1 -2246.483,E2 -2246.483} C_VEL
LIN {X 0,Y 572.959,Z 327.806,A -85,B 0,C 180,E1 -2247.187,E2 -2247.187} C_VEL
LIN {X 0,Y 572.94,Z 329.196,A -85,B 0,C 180,E1 -2247.89,E2 -2247.89} C_VEL
LIN {X 0,Y 572.941,Z 330.784,A -85,B 0,C 180,E1 -2249.296,E2 -2249.296} C_VEL
LIN {X 0,Y 572.938,Z 331,A -85,B 0,C 180,E1 -2249.999,E2 -2249.999} C_VEL
LIN {X 0,Y 572.946,Z 330.187,A -85,B 0,C 180,E1 -2251.405,E2 -2251.405} C_VEL
LIN {X 0,Y 572.94,Z 329.201,A -85,B 0,C 180,E1 -2252.108,E2 -2252.108} C_VEL
LIN {X 0,Y 572.959,Z 327.813,A -85,B 0,C 180,E1 -2252.811,E2 -2252.811} C_VEL
LIN {X 0,Y 573.014,Z 324.9,A -85,B 0,C 180,E1 -2253.867,E2 -2253.867} C_VEL
LIN {X 0,Y 572.963,Z 320.954,A -85,B 0,C 180,E1 -2254.924,E2 -2254.924} C_VEL
LIN {X 0,Y 573.097,Z 315.873,A -85,B 0,C 180,E1 -2255.982,E2 -2255.982} C_VEL
LIN {X 0,Y 573.103,Z 309.476,A -85,B 0,C 180,E1 -2257.043,E2 -2257.043} C_VEL
LIN {X 0,Y 573.177,Z 301.489,A -85,B 0,C 180,E1 -2258.105,E2 -2258.105} C_VEL
LIN {X 0,Y 573.253,Z 293.348,A -85,B 0,C 180,E1 -2258.992,E2 -2258.992} C_VEL
LIN {X 0,Y 573.345,Z 283.416,A -85,B 0,C 180,E1 -2259.88,E2 -2259.88} C_VEL
LIN {X 0,Y 573.503,Z 272.23,A -85,B 0,C 180,E1 -2260.678,E2 -2260.678} C_VEL
LIN {X 0,Y 573.578,Z 261.201,A -85,B 0,C 180,E1 -2261.305,E2 -2261.305} C_VEL
LIN {X 0,Y 573.695,Z 249.015,A -85,B 0,C 180,E1 -2261.839,E2 -2261.839} C_VEL
LIN {X 0,Y 573.807,Z 236.228,A -85,B 0,C 180,E1 -2262.241,E2 -2262.241} C_VEL
LIN {X 0,Y 573.838,Z 224.946,A -85,B 0,C 180,E1 -2262.476,E2 -2262.476} C_VEL
LIN {X 0,Y 573.22,Z 220.818,A -85,B 0,C 180,E1 -2262.568,E2 -2262.568} C_VEL
LIN {X 0,Y 573.321,Z 205.618,A -85,B 0,C 180,E1 -2265.28,E2 -2265.28} C_VEL
LIN {X 0,Y 573.474,Z 190.418,A -85,B 0,C 180,E1 -2268.024,E2 -2268.024} C_VEL
LIN {X 0,Y 573.605,Z 175.227,A -85,B 0,C 180,E1 -2270.811,E2 -2270.811} C_VEL
LIN {X 0,Y 573.797,Z 162.061,A -85,B 0,C 180,E1 -2273.275,E2 -2273.275} C_VEL
LIN {X 0,Y 574.002,Z 146.993,A -85,B 0,C 180,E1 -2276.152,E2 -2276.152} C_VEL
LIN {X 0,Y 573.45,Z 141.968,A -85,B 0,C 180,E1 -2277.161,E2 -2277.161} C_VEL
LIN {X 0,Y 573.263,Z 141.08,A -85,B 0,C 180,E1 -2277.368,E2 -2277.368} C_VEL
LIN {X 0,Y 573.222,Z 141.082,A -85,B 0,C 180,E1 -2280.176,E2 -2280.176} C_VEL
LIN {X 0,Y 573.25,Z 141.08,A -85,B 0,C 180,E1 -2282.644,E2 -2282.644} C_VEL
LIN {X 0,Y 573.265,Z 141.075,A -85,B 0,C 180,E1 -2285.182,E2 -2285.182} C_VEL
LIN {X 0,Y 573.229,Z 141.081,A -85,B 0,C 180,E1 -2287.806,E2 -2287.806} C_VEL
LIN {X 0,Y 573.236,Z 141.081,A -85,B 0,C 180,E1 -2290.524,E2 -2290.524} C_VEL
LIN {X 0,Y 573.22,Z 141.079,A -85,B 0,C 180,E1 -2293.359,E2 -2293.359} C_VEL
LIN {X 0,Y 573.244,Z 141.078,A -85,B 0,C 180,E1 -2296.329,E2 -2296.329} C_VEL
LIN {X 0,Y 573.264,Z 141.078,A -85,B 0,C 180,E1 -2299.476,E2 -2299.476} C_VEL
LIN {X 0,Y 573.221,Z 141.082,A -85,B 0,C 180,E1 -2302.191,E2 -2302.191} C_VEL
LIN {X 0,Y 573.212,Z 141.08,A -85,B 0,C 180,E1 -2305.229,E2 -2305.229} C_VEL
LIN {X 0,Y 573.247,Z 141.081,A -85,B 0,C 180,E1 -2307.769,E2 -2307.769} C_VEL
LIN {X 0,Y 573.259,Z 141.078,A -85,B 0,C 180,E1 -2310.634,E2 -2310.634} C_VEL
LIN {X 0,Y 573.26,Z 141.075,A -85,B 0,C 180,E1 -2313.499,E2 -2313.499} C_VEL
LIN {X 0,Y 573.214,Z 141.085,A -85,B 0,C 180,E1 -2316.134,E2 -2316.134} C_VEL
LIN {X 0,Y 573.238,Z 141.082,A -85,B 0,C 180,E1 -2319.173,E2 -2319.173} C_VEL
LIN {X 0,Y 573.229,Z 141.081,A -85,B 0,C 180,E1 -2321.411,E2 -2321.411} C_VEL
LIN {X 0,Y 573.249,Z 141.076,A -85,B 0,C 180,E1 -2323.622,E2 -2323.622} C_VEL
LIN {X 0,Y 573.271,Z 141.077,A -85,B 0,C 180,E1 -2325.807,E2 -2325.807} C_VEL
LIN {X 0,Y 573.246,Z 141.076,A -85,B 0,C 180,E1 -2328.745,E2 -2328.745} C_VEL
LIN {X 0,Y 573.259,Z 141.076,A -85,B 0,C 180,E1 -2331.54,E2 -2331.54} C_VEL
LIN {X 0,Y 573.281,Z 141.078,A -85,B 0,C 180,E1 -2334.372,E2 -2334.372} C_VEL
LIN {X 0,Y 573.299,Z 141.076,A -85,B 0,C 180,E1 -2337.892,E2 -2337.892} C_VEL
LIN {X 0,Y 573.316,Z 141.069,A -85,B 0,C 180,E1 -2340.702,E2 -2340.702} C_VEL
LIN {X 0,Y 573.207,Z 141.081,A -85,B 0,C 180,E1 -2343.515,E2 -2343.515} C_VEL
LIN {X 0,Y 573.274,Z 141.074,A -85,B 0,C 180,E1 -2345.628,E2 -2345.628} C_VEL
LIN {X 0,Y 573.298,Z 141.071,A -85,B 0,C 180,E1 -2348.459,E2 -2348.459} C_VEL
LIN {X 0,Y 573.284,Z 141.078,A -85,B 0,C 180,E1 -2351.312,E2 -2351.312} C_VEL
LIN {X 0,Y 573.259,Z 141.079,A -85,B 0,C 180,E1 -2354.422,E2 -2354.422} C_VEL
LIN {X 0,Y 573.246,Z 141.076,A -85,B 0,C 180,E1 -2357.112,E2 -2357.112} C_VEL
LIN {X 0,Y 573.245,Z 141.078,A -85,B 0,C 180,E1 -2360.077,E2 -2360.077} C_VEL
LIN {X 0,Y 573.258,Z 141.08,A -85,B 0,C 180,E1 -2363.154,E2 -2363.154} C_VEL
LIN {X 0,Y 573.241,Z 141.081,A -85,B 0,C 180,E1 -2364.407,E2 -2364.407} C_VEL
LIN {X 0,Y 572.601,Z 141.165,A -85,B 0,C 180,E1 -2364.994,E2 -2364.994} C_VEL
LIN {X 0,Y 569.734,Z 141.521,A -85,B 0,C 180,E1 -2365.945,E2 -2365.945} C_VEL
LIN {X 0,Y 567.289,Z 141.82,A -85,B 0,C 180,E1 -2366.71,E2 -2366.71} C_VEL
LIN {X 0,Y 566.235,Z 141.949,A -85,B 0,C 180,E1 -2367.301,E2 -2367.301} C_VEL
LIN {X 0,Y 566.149,Z 141.96,A -85,B 0,C 180,E1 -2367.502,E2 -2367.502} C_VEL
LIN {X 0,Y 566.191,Z 141.962,A -85,B 0,C 180,E1 -2369.769,E2 -2369.769} C_VEL
LIN {X 0,Y 566.195,Z 141.955,A -85,B 0,C 180,E1 -2372.432,E2 -2372.432} C_VEL
LIN {X 0,Y 566.205,Z 141.957,A -85,B 0,C 180,E1 -2374.996,E2 -2374.996} C_VEL
LIN {X 0,Y 566.185,Z 141.957,A -85,B 0,C 180,E1 -2377.462,E2 -2377.462} C_VEL
